  MoveL 10167 to (522.4, 527.74, 184) mm, rotated rx -180 ry 0 rz 160 deg; joints [9.235, 54.746, -7.823, -142.539, 53.417, 155.455]
  Set speed (17.9 mm/s)
  Call Extruder(893.93163)
  MoveL 10168 to (521.41, 528.51, 184) mm, rotated rx 180 ry 0 rz 160 deg; joints [9.346, 54.585, -7.526, -142.475, 53.571, 155.484]
  Set speed (17.9 mm/s)
  Call Extruder(896.88421)
  MoveL 10169 to (520.65, 529.06, 184) mm, rotated rx -180 ry 0 rz 160 deg; joints [9.426, 54.462, -7.298, -142.432, 53.688, 155.51]
  Call Extruder(901.40874)
  MoveL 10170 to (519.47, 529.87, 184) mm, rotated rx 180 ry 0 rz 160 deg; joints [9.545, 54.269, -6.939, -142.372, 53.869, 155.556]
  Call Extruder(903.78888)
  MoveL 10171 to (518.83, 530.27, 184) mm, rotated rx 180 ry 0 rz 160 deg; joints [9.606, 54.164, -6.745, -142.343, 53.965, 155.583]
  Set speed (17.9 mm/s)
  Call Extruder(906.07988)
  MoveL 10172 to (518.21, 530.65, 184) mm, rotated rx 180 ry 0 rz 160 deg; joints [9.663, 54.063, -6.556, -142.317, 54.057, 155.611]
  Call Extruder(910.83041)
  MoveL 10173 to (516.91, 531.39, 184) mm, rotated rx 180 ry 0 rz 160 deg; joints [9.779, 53.847, -6.156, -142.269, 54.25, 155.674]
  Set speed (17.8 mm/s)
  Call Extruder(914.28684)
  MoveL 10174 to (515.94, 531.89, 184) mm, rotated rx 180 ry 0 rz 160 deg; joints [9.859, 53.687, -5.859, -142.239, 54.392, 155.725]
  Call Extruder(917.59208)
  MoveL 10175 to (515, 532.34, 184) mm, rotated rx 180 ry 0 rz 160 deg; joints [9.933, 53.53, -5.568, -142.215, 54.528, 155.778]
  Set speed (17.9 mm/s)
  Call Extruder(922.23001)
  MoveL 10176 to (513.65, 532.93, 184) mm, rotated rx -180 ry 0 rz 160 deg; joints [10.032, 53.306, -5.154, -142.187, 54.719, 155.857]
  Set speed (17.9 mm/s)
  Call Extruder(926.66688)
  MoveL 10177 to (512.34, 533.45, 184) mm, rotated rx 180 ry 0 rz 160 deg; joints [10.121, 53.088, -4.749, -142.168, 54.903, 155.939]
  Set speed (17.8 mm/s)
  Call Extruder(929.18658)
  MoveL 10178 to (511.59, 533.71, 184) mm, rotated rx -180 ry 0 rz 160 deg; joints [10.169, 52.962, -4.515, -142.161, 55.008, 155.989]
  Set speed (17.8 mm/s)
  Call Extruder(932.98840)
  MoveL 10179 to (510.45, 534.08, 184) mm, rotated rx 180 ry 0 rz 160 deg; joints [10.239, 52.771, -4.161, -142.153, 55.165, 156.067]
  Set speed (17.8 mm/s)
  Call Extruder(936.81967)
  MoveL 10180 to (509.29, 534.42, 184) mm, rotated rx -180 ry 0 rz 160 deg; joints [10.305, 52.576, -3.799, -142.15, 55.323, 156.149]
  Set speed (17.8 mm/s)
  Call Extruder(940.52296)
  MoveL 10181 to (508.15, 534.7, 184) mm, rotated rx -180 ry 0 rz 160 deg; joints [10.364, 52.384, -3.444, -142.153, 55.476, 156.233]
  Set speed (17.9 mm/s)
  Call Extruder(945.30301)
  MoveL 10182 to (506.68, 535.02, 184) mm, rotated rx -180 ry 0 rz 160 deg; joints [10.436, 52.134, -2.982, -142.163, 55.673, 156.347]
  Call Extruder(949.97825)
  MoveL 10183 to (505.22, 535.27, 184) mm, rotated rx -180 ry 0 rz 160 deg; joints [10.498, 51.886, -2.524, -142.182, 55.864, 156.464]
  Set speed (17.8 mm/s)
  Call Extruder(954.40667)
  MoveL 10184 to (503.83, 535.45, 184) mm, rotated rx 180 ry 0 rz 160 deg; joints [10.552, 51.65, -2.087, -142.206, 56.044, 156.579]
  Set speed (17.9 mm/s)
  Call Extruder(959.14962)
  MoveL 10185 to (502.33, 535.57, 184) mm, rotated rx -180 ry 0 rz 160 deg; joints [10.602, 51.396, -1.616, -142.24, 56.235, 156.708]
  Set speed (17.9 mm/s)
  Call Extruder(963.82186)
  MoveL 10186 to (500.86, 535.64, 184) mm, rotated rx 180 ry 0 rz 160 deg; joints [10.644, 51.143, -1.149, -142.281, 56.421, 156.84]
  Set speed (17.9 mm/s)
  Call Extruder(968.31975)
  MoveL 10187 to (499.43, 535.65, 184) mm, rotated rx 180 ry 0 rz 160 deg; joints [10.678, 50.899, -0.698, -142.327, 56.598, 156.971]
  Set speed (10.0 mm/s)
  MoveL 10188 to (499.43, 535.65, 188) mm, rotated rx -180 ry 0 rz 160 deg; joints [10.678, 50.375, -0.656, -142.13, 56.216, 156.616]
  Set speed (120.0 mm/s)
  MoveL 10189 to (500.85, 535.22, 188) mm, rotated rx -180 ry 0 rz 160 deg; joints [10.593, 50.605, -1.079, -142.145, 56.03, 156.526]
  Set speed (18.0 mm/s)
  Call Extruder(972.66654)
  MoveL 10190 to (499.46, 535.23, 188) mm, rotated rx 180 ry 0 rz 160 deg; joints [10.625, 50.366, -0.641, -142.191, 56.201, 156.653]
  Call Extruder(977.34606)
  MoveL 10191 to (497.97, 535.17, 188) mm, rotated rx -180 ry 0 rz 160 deg; joints [10.653, 50.109, -0.168, -142.248, 56.382, 156.795]
  Set speed (18.0 mm/s)
  Call Extruder(981.88642)
  MoveL 10192 to (496.53, 535.06, 188) mm, rotated rx -180 ry 0 rz 160 deg; joints [10.673, 49.859, 0.291, -142.311, 56.555, 156.936]
  Call Extruder(986.34744)
  MoveL 10193 to (495.12, 534.89, 188) mm, rotated rx 180 ry 0 rz 160 deg; joints [10.685, 49.613, 0.741, -142.38, 56.722, 157.078]
  Set speed (18.0 mm/s)
  Call Extruder(990.84090)
  MoveL 10194 to (493.71, 534.67, 188) mm, rotated rx -180 ry 0 rz 160 deg; joints [10.69, 49.367, 1.192, -142.457, 56.886, 157.225]
  Set speed (18.0 mm/s)
  Call Extruder(995.48981)
  MoveL 10195 to (492.26, 534.37, 188) mm, rotated rx 180 ry 0 rz 160 deg; joints [10.687, 49.113, 1.658, -142.544, 57.053, 157.38]
  Set speed (18.0 mm/s)
  Call Extruder(999.88346)
  MoveL 10196 to (490.9, 534.04, 188) mm, rotated rx 180 ry 0 rz 160 deg; joints [10.678, 48.874, 2.095, -142.632, 57.207, 157.53]
  Set speed (18.0 mm/s)
  Call Extruder(1004.84592)
  MoveL 10197 to (489.39, 533.6, 188) mm, rotated rx 180 ry 0 rz 160 deg; joints [10.658, 48.607, 2.585, -142.74, 57.376, 157.702]
  Set speed (18.0 mm/s)
  Call Extruder(1008.82941)
  MoveL 10198 to (488.18, 533.19, 188) mm, rotated rx 180 ry 0 rz 160 deg; joints [10.635, 48.394, 2.974, -142.833, 57.509, 157.842]
  Set speed (18.0 mm/s)
  Call Extruder(1013.42678)
  MoveL 10199 to (486.82, 532.67, 188) mm, rotated rx 180 ry 0 rz 160 deg; joints [10.602, 48.151, 3.419, -142.947, 57.657, 158.005]
  Set speed (18.0 mm/s)
  Call Extruder(1017.94180)
  MoveL 10200 to (485.49, 532.11, 188) mm, rotated rx -180 ry 0 rz 160 deg; joints [10.562, 47.915, 3.851, -143.066, 57.798, 158.168]
  Set speed (17.9 mm/s)
  Call Extruder(1021.37830)
  MoveL 10201 to (484.5, 531.64, 188) mm, rotated rx -180 ry 0 rz 160 deg; joints [10.526, 47.738, 4.174, -143.16, 57.902, 158.293]
  Set speed (18.0 mm/s)
  Call Extruder(1024.92138)
  MoveL 10202 to (483.5, 531.14, 188) mm, rotated rx 180 ry 0 rz 160 deg; joints [10.485, 47.557, 4.505, -143.261, 58.007, 158.423]
  Set speed (18.0 mm/s)
  Call Extruder(1029.79745)
  MoveL 10203 to (482.14, 530.37, 188) mm, rotated rx 180 ry 0 rz 160 deg; joints [10.419, 47.313, 4.952, -143.408, 58.145, 158.603]
  Set speed (18.0 mm/s)
  Call Extruder(1034.30455)
  MoveL 10204 to (480.92, 529.62, 188) mm, rotated rx 180 ry 0 rz 160 deg; joints [10.351, 47.091, 5.356, -143.551, 58.267, 158.771]
  Call Extruder(1038.31068)
  MoveL 10205 to (479.86, 528.91, 188) mm, rotated rx -180 ry 0 rz 160 deg; joints [10.284, 46.898, 5.709, -143.682, 58.371, 158.92]
  Set speed (18.0 mm/s)
  Call Extruder(1040.61575)
  MoveL 10206 to (479.26, 528.48, 188) mm, rotated rx 180 ry 0 rz 160 deg; joints [10.243, 46.788, 5.909, -143.76, 58.43, 159.006]
  Set speed (18.0 mm/s)
  Call Extruder(1042.87029)
  MoveL 10207 to (478.69, 528.06, 188) mm, rotated rx 180 ry 0 rz 160 deg; joints [10.201, 46.682, 6.102, -143.838, 58.485, 159.091]
  Call Extruder(1045.13772)
  MoveL 10208 to (478.12, 527.61, 188) mm, rotated rx -180 ry 0 rz 160 deg; joints [10.157, 46.577, 6.294, -143.918, 58.539, 159.176]
  Set speed (18.0 mm/s)
  Call Extruder(1047.91484)
  MoveL 10209 to (477.43, 527.06, 188) mm, rotated rx 180 ry 0 rz 160 deg; joints [10.1, 46.45, 6.525, -144.017, 58.604, 159.281]
  Set speed (18.0 mm/s)
  Call Extruder(1050.88641)
  MoveL 10210 to (476.71, 526.44, 188) mm, rotated rx -180 ry 0 rz 160 deg; joints [10.037, 46.317, 6.768, -144.126, 58.67, 159.392]
  Set speed (18.0 mm/s)
  Call Extruder(1054.07637)
  MoveL 10211 to (475.96, 525.76, 188) mm, rotated rx 180 ry 0 rz 160 deg; joints [9.965, 46.177, 7.023, -144.246, 58.738, 159.512]
  Set speed (18.0 mm/s)
  Call Extruder(1056.93409)
  MoveL 10212 to (475.31, 525.13, 188) mm, rotated rx -180 ry 0 rz 160 deg; joints [9.898, 46.054, 7.247, -144.355, 58.797, 159.619]
  Set speed (18.0 mm/s)
  Call Extruder(1060.97638)
  MoveL 10213 to (474.4, 524.21, 188) mm, rotated rx -180 ry 0 rz 160 deg; joints [9.798, 45.884, 7.557, -144.514, 58.876, 159.771]
  Set speed (18.0 mm/s)
  Call Extruder(1063.75696)
  MoveL 10214 to (473.8, 523.56, 188) mm, rotated rx 180 ry 0 rz 160 deg; joints [9.726, 45.77, 7.764, -144.626, 58.927, 159.875]
  Set speed (18.0 mm/s)
  Call Extruder(1066.38918)
  MoveL 10215 to (473.25, 522.93, 188) mm, rotated rx -180 ry 0 rz 160 deg; joints [9.655, 45.664, 7.957, -144.733, 58.974, 159.973]
  Call Extruder(1070.04487)
  MoveL 10216 to (472.51, 522.03, 188) mm, rotated rx 180 ry 0 rz 160 deg; joints [9.554, 45.522, 8.216, -144.885, 59.034, 160.109]
  Set speed (18.0 mm/s)
  Call Extruder(1074.65991)
  MoveL 10217 to (471.61, 520.87, 188) mm, rotated rx 180 ry 0 rz 160 deg; joints [9.419, 45.348, 8.532, -145.081, 59.105, 160.28]
  Set speed (18.0 mm/s)
  Call Extruder(1076.75495)
  MoveL 10218 to (471.22, 520.33, 188) mm, rotated rx -180 ry 0 rz 160 deg; joints [9.356, 45.272, 8.67, -145.172, 59.135, 160.357]
  Set speed (18.0 mm/s)
  Call Extruder(1079.16479)
  MoveL 10219 to (470.78, 519.69, 188) mm, rotated rx 180 ry 0 rz 160 deg; joints [9.282, 45.187, 8.826, -145.277, 59.168, 160.445]
  Set speed (18.0 mm/s)
  Call Extruder(1081.78892)
  MoveL 10220 to (470.33, 519, 188) mm, rotated rx 180 ry 0 rz 160 deg; joints [9.199, 45.096, 8.991, -145.393, 59.201, 160.541]
  Set speed (18.0 mm/s)
  Call Extruder(1083.58163)
  MoveL 10221 to (470.02, 518.51, 188) mm, rotated rx -180 ry 0 rz 160 deg; joints [9.141, 45.036, 9.1, -145.474, 59.222, 160.606]
  Set speed (18.0 mm/s)
  Call Extruder(1086.37228)
  MoveL 10222 to (469.57, 517.75, 188) mm, rotated rx 180 ry 0 rz 160 deg; joints [9.049, 44.944, 9.267, -145.6, 59.254, 160.707]
  Set speed (18.0 mm/s)
  Call Extruder(1090.55089)
  MoveL 10223 to (468.91, 516.59, 188) mm, rotated rx -180 ry 0 rz 160 deg; joints [8.908, 44.812, 9.506, -145.791, 59.296, 160.857]
  Call Extruder(1092.71321)
  MoveL 10224 to (468.6, 515.98, 188) mm, rotated rx 180 ry 0 rz 160 deg; joints [8.833, 44.747, 9.625, -145.891, 59.315, 160.934]
  Set speed (18.0 mm/s)
  Call Extruder(1094.90666)
  MoveL 10225 to (468.29, 515.35, 188) mm, rotated rx -180 ry 0 rz 160 deg; joints [8.755, 44.683, 9.741, -145.994, 59.334, 161.011]
  Call Extruder(1099.61642)
  MoveL 10226 to (467.66, 513.99, 188) mm, rotated rx 180 ry 0 rz 160 deg; joints [8.585, 44.552, 9.979, -146.216, 59.367, 161.176]
  Call Extruder(1103.98776)
  MoveL 10227 to (467.14, 512.7, 188) mm, rotated rx 180 ry 0 rz 160 deg; joints [8.423, 44.439, 10.185, -146.425, 59.392, 161.327]
  Set speed (18.0 mm/s)
  Call Extruder(1108.45870)
  MoveL 10228 to (466.65, 511.36, 188) mm, rotated rx -180 ry 0 rz 160 deg; joints [8.252, 44.332, 10.379, -146.642, 59.41, 161.478]
  Set speed (18.0 mm/s)
  Call Extruder(1110.08883)
  MoveL 10229 to (466.49, 510.87, 188) mm, rotated rx 180 ry 0 rz 160 deg; joints [8.189, 44.295, 10.446, -146.721, 59.415, 161.533]
  Set speed (17.9 mm/s)
  Call Extruder(1113.55157)
  MoveL 10230 to (466.16, 509.82, 188) mm, rotated rx 180 ry 0 rz 160 deg; joints [8.053, 44.22, 10.581, -146.891, 59.423, 161.648]
  Set speed (18.0 mm/s)
  Call Extruder(1117.54079)
  MoveL 10231 to (465.83, 508.59, 188) mm, rotated rx -180 ry 0 rz 160 deg; joints [7.893, 44.141, 10.724, -147.087, 59.427, 161.778]
  Set speed (18.0 mm/s)
  Call Extruder(1122.08861)
  MoveL 10232 to (465.51, 507.18, 188) mm, rotated rx 180 ry 0 rz 160 deg; joints [7.708, 44.06, 10.871, -147.313, 59.425, 161.923]
  Set speed (18.0 mm/s)
  Call Extruder(1126.74925)
  MoveL 10233 to (465.23, 505.72, 188) mm, rotated rx -180 ry 0 rz 160 deg; joints [7.515, 43.987, 11.004, -147.545, 59.415, 162.069]
  Set speed (18.0 mm/s)
  Call Extruder(1131.27133)
  MoveL 10234 to (465.03, 504.3, 188) mm, rotated rx 180 ry 0 rz 160 deg; joints [7.325, 43.926, 11.115, -147.771, 59.399, 162.207]
  Call Extruder(1135.79933)
  MoveL 10235 to (464.88, 502.87, 188) mm, rotated rx 180 ry 0 rz 160 deg; joints [7.132, 43.875, 11.208, -147.997, 59.375, 162.341]
  Call Extruder(1140.43813)
  MoveL 10236 to (464.8, 501.39, 188) mm, rotated rx -180 ry 0 rz 160 deg; joints [6.933, 43.832, 11.284, -148.229, 59.344, 162.475]
  Set speed (17.9 mm/s)
  Call Extruder(1144.77516)
  MoveL 10237 to (464.77, 500.01, 188) mm, rotated rx -180 ry 0 rz 160 deg; joints [6.745, 43.802, 11.339, -148.445, 59.309, 162.596]
  Set speed (17.9 mm/s)
  Call Extruder(1148.91787)
  MoveL 10238 to (464.79, 498.69, 188) mm, rotated rx 180 ry 0 rz 160 deg; joints [6.565, 43.782, 11.376, -148.65, 59.269, 162.708]
  Set speed (18.0 mm/s)
  Call Extruder(1152.91329)
  MoveL 10239 to (464.86, 497.43, 188) mm, rotated rx 180 ry 0 rz 160 deg; joints [6.39, 43.77, 11.397, -148.847, 59.226, 162.813]
  Set speed (18.0 mm/s)
  Call Extruder(1156.99605)
  MoveL 10240 to (464.98, 496.13, 188) mm, rotated rx 180 ry 0 rz 160 deg; joints [6.211, 43.766, 11.404, -149.047, 59.176, 162.917]
  Set speed (18.0 mm/s)
  Call Extruder(1161.07084)
  MoveL 10241 to (465.15, 494.84, 188) mm, rotated rx 180 ry 0 rz 160 deg; joints [6.033, 43.771, 11.396, -149.244, 59.12, 163.017]
  Call Extruder(1164.98026)
  MoveL 10242 to (465.35, 493.61, 188) mm, rotated rx -180 ry 0 rz 160 deg; joints [5.862, 43.783, 11.374, -149.432, 59.062, 163.109]
  Set speed (18.0 mm/s)
  Call Extruder(1169.18292)
  MoveL 10243 to (465.62, 492.3, 188) mm, rotated rx 180 ry 0 rz 160 deg; joints [5.679, 43.804, 11.336, -149.631, 58.994, 163.204]
  Set speed (18.0 mm/s)
  Call Extruder(1173.28818)
  MoveL 10244 to (465.93, 491.03, 188) mm, rotated rx -180 ry 0 rz 160 deg; joints [5.502, 43.833, 11.284, -149.822, 58.923, 163.292]
  Set speed (18.0 mm/s)
  Call Extruder(1177.30378)
  MoveL 10245 to (466.27, 489.8, 188) mm, rotated rx 180 ry 0 rz 160 deg; joints [5.329, 43.869, 11.218, -150.007, 58.848, 163.375]
  Set speed (18.0 mm/s)
  Call Extruder(1181.38217)
  MoveL 10246 to (466.67, 488.57, 188) mm, rotated rx 180 ry 0 rz 160 deg; joints [5.155, 43.914, 11.137, -150.19, 58.767, 163.454]
  Call Extruder(1185.55335)
  MoveL 10247 to (467.13, 487.32, 188) mm, rotated rx -180 ry 0 rz 160 deg; joints [4.979, 43.968, 11.038, -150.375, 58.678, 163.531]
  Set speed (18.0 mm/s)
  Call Extruder(1189.67180)
  MoveL 10248 to (467.62, 486.11, 188) mm, rotated rx -180 ry 0 rz 160 deg; joints [4.807, 44.03, 10.927, -150.552, 58.586, 163.603]
  Set speed (18.0 mm/s)
  Call Extruder(1193.68830)
  MoveL 10249 to (468.15, 484.94, 188) mm, rotated rx 180 ry 0 rz 160 deg; joints [4.642, 44.097, 10.805, -150.721, 58.492, 163.668]
  Set speed (18.0 mm/s)
  Call Extruder(1197.78489)
  MoveL 10250 to (468.73, 483.77, 188) mm, rotated rx 180 ry 0 rz 160 deg; joints [4.477, 44.174, 10.665, -150.889, 58.391, 163.73]
  Set speed (18.0 mm/s)
  Call Extruder(1201.93796)
  MoveL 10251 to (469.36, 482.61, 188) mm, rotated rx 180 ry 0 rz 160 deg; joints [4.312, 44.259, 10.51, -151.054, 58.284, 163.788]
  Set speed (17.9 mm/s)
  Call Extruder(1206.52795)
  MoveL 10252 to (470.1, 481.36, 188) mm, rotated rx 180 ry 0 rz 160 deg; joints [4.134, 44.363, 10.323, -151.23, 58.161, 163.846]
  Set speed (18.0 mm/s)
  Call Extruder(1209.83621)
  MoveL 10253 to (470.68, 480.47, 188) mm, rotated rx -180 ry 0 rz 160 deg; joints [4.008, 44.443, 10.176, -151.353, 58.068, 163.884]
  Set speed (18.0 mm/s)
  Call Extruder(1214.03556)
  MoveL 10254 to (471.44, 479.37, 188) mm, rotated rx -180 ry 0 rz 160 deg; joints [3.852, 44.552, 9.978, -151.503, 57.947, 163.928]
  Set speed (18.0 mm/s)
  Call Extruder(1218.05006)
  MoveL 10255 to (472.21, 478.35, 188) mm, rotated rx -180 ry 0 rz 160 deg; joints [3.707, 44.664, 9.776, -151.641, 57.827, 163.964]
  Call Extruder(1222.27088)
  MoveL 10256 to (473.05, 477.31, 188) mm, rotated rx 180 ry 0 rz 160 deg; joints [3.558, 44.788, 9.551, -151.779, 57.696, 163.997]
  Set speed (18.0 mm/s)
  Call Extruder(1226.25255)
  MoveL 10257 to (473.88, 476.35, 188) mm, rotated rx 180 ry 0 rz 160 deg; joints [3.423, 44.911, 9.326, -151.904, 57.57, 164.024]
  Call Extruder(1230.41361)
  MoveL 10258 to (474.79, 475.39, 188) mm, rotated rx -180 ry 0 rz 160 deg; joints [3.285, 45.047, 9.079, -152.027, 57.434, 164.046]
  Set speed (18.0 mm/s)
  Call Extruder(1234.40312)
  MoveL 10259 to (475.7, 474.49, 188) mm, rotated rx 180 ry 0 rz 160 deg; joints [3.158, 45.184, 8.83, -152.138, 57.3, 164.062]
  Set speed (18.0 mm/s)
  Call Extruder(1238.47932)
  MoveL 10260 to (476.65, 473.62, 188) mm, rotated rx 180 ry 0 rz 160 deg; joints [3.034, 45.33, 8.565, -152.245, 57.16, 164.073]
  Set speed (18.0 mm/s)
  Call Extruder(1242.64814)
  MoveL 10261 to (477.66, 472.75, 188) mm, rotated rx -180 ry 0 rz 160 deg; joints [2.911, 45.485, 8.282, -152.347, 57.014, 164.078]
  Set speed (18.0 mm/s)
  Call Extruder(1247.06946)
  MoveL 10262 to (478.77, 471.88, 188) mm, rotated rx -180 ry 0 rz 160 deg; joints [2.788, 45.657, 7.97, -152.446, 56.856, 164.078]
  Call Extruder(1250.74658)
  MoveL 10263 to (479.71, 471.2, 188) mm, rotated rx 180 ry 0 rz 160 deg; joints [2.69, 45.805, 7.701, -152.522, 56.721, 164.073]
  Set speed (18.0 mm/s)
  Call Extruder(1254.67182)
  MoveL 10264 to (480.75, 470.49, 188) mm, rotated rx -180 ry 0 rz 160 deg; joints [2.59, 45.967, 7.405, -152.597, 56.576, 164.062]
  Call Extruder(1258.92817)
  MoveL 10265 to (481.9, 469.78, 188) mm, rotated rx 180 ry 0 rz 160 deg; joints [2.488, 46.149, 7.074, -152.669, 56.415, 164.045]
  Call Extruder(1263.01389)
  MoveL 10266 to (483.02, 469.13, 188) mm, rotated rx 180 ry 0 rz 160 deg; joints [2.396, 46.329, 6.747, -152.73, 56.258, 164.023]
  Set speed (18.0 mm/s)
  Call Extruder(1266.90627)
  MoveL 10267 to (484.12, 468.55, 188) mm, rotated rx 180 ry 0 rz 160 deg; joints [2.313, 46.504, 6.427, -152.781, 56.107, 163.996]
  Set speed (18.0 mm/s)
  Call Extruder(1271.14857)
  MoveL 10268 to (485.34, 467.96, 188) mm, rotated rx 180 ry 0 rz 160 deg; joints [2.23, 46.7, 6.07, -152.828, 55.941, 163.961]
  Set speed (18.0 mm/s)
  Call Extruder(1275.23430)
  MoveL 10269 to (486.53, 467.45, 188) mm, rotated rx 180 ry 0 rz 160 deg; joints [2.155, 46.893, 5.718, -152.866, 55.779, 163.922]
  Set speed (18.0 mm/s)
  Call Extruder(1279.11549)
  MoveL 10270 to (487.68, 466.99, 188) mm, rotated rx 180 ry 0 rz 160 deg; joints [2.09, 47.08, 5.376, -152.893, 55.623, 163.88]
  Set speed (18.0 mm/s)
  Call Extruder(1283.35551)
  MoveL 10271 to (488.95, 466.54, 188) mm, rotated rx -180 ry 0 rz 160 deg; joints [2.026, 47.288, 4.996, -152.914, 55.452, 163.827]
  Call Extruder(1287.41205)
  MoveL 10272 to (490.19, 466.16, 188) mm, rotated rx 180 ry 0 rz 160 deg; joints [1.971, 47.491, 4.626, -152.926, 55.288, 163.771]
  Set speed (18.0 mm/s)
  Call Extruder(1291.52994)
  MoveL 10273 to (491.45, 465.82, 188) mm, rotated rx 180 ry 0 rz 160 deg; joints [1.921, 47.7, 4.244, -152.93, 55.12, 163.708]
  Call Extruder(1295.44431)
  MoveL 10274 to (492.67, 465.54, 188) mm, rotated rx -180 ry 0 rz 160 deg; joints [1.879, 47.902, 3.875, -152.926, 54.959, 163.644]
  Call Extruder(1299.59154)
  MoveL 10275 to (493.96, 465.29, 188) mm, rotated rx 180 ry 0 rz 160 deg; joints [1.841, 48.118, 3.48, -152.913, 54.789, 163.57]
  Set speed (18.0 mm/s)
  Call Extruder(1303.53526)
  MoveL 10276 to (495.2, 465.09, 188) mm, rotated rx 180 ry 0 rz 160 deg; joints [1.811, 48.326, 3.099, -152.893, 54.627, 163.494]
  Set speed (18.0 mm/s)
  Call Extruder(1307.77538)
  MoveL 10277 to (496.55, 464.94, 188) mm, rotated rx 180 ry 0 rz 160 deg; joints [1.785, 48.552, 2.686, -152.862, 54.452, 163.406]
  Call Extruder(1311.80226)
  MoveL 10278 to (497.82, 464.84, 188) mm, rotated rx 180 ry 0 rz 160 deg; joints [1.767, 48.768, 2.289, -152.825, 54.287, 163.318]
  Set speed (18.0 mm/s)
  Call Extruder(1315.97904)
  MoveL 10279 to (499.15, 464.78, 188) mm, rotated rx 180 ry 0 rz 160 deg; joints [1.755, 48.995, 1.875, -152.777, 54.116, 163.22]
  Set speed (18.0 mm/s)
  Call Extruder(1319.97418)
  MoveL 10280 to (500.42, 464.77, 188) mm, rotated rx -180 ry 0 rz 160 deg; joints [1.748, 49.212, 1.476, -152.724, 53.953, 163.122]
  Call Extruder(1324.11243)
  MoveL 10281 to (501.74, 464.81, 188) mm, rotated rx 180 ry 0 rz 160 deg; joints [1.748, 49.439, 1.061, -152.661, 53.786, 163.015]
  Set speed (18.0 mm/s)
  Call Extruder(1328.11577)
  MoveL 10282 to (503.01, 464.9, 188) mm, rotated rx -180 ry 0 rz 160 deg; joints [1.754, 49.658, 0.658, -152.592, 53.625, 162.906]
  Set speed (18.0 mm/s)
  Call Extruder(1332.26885)
  MoveL 10283 to (504.33, 465.04, 188) mm, rotated rx -180 ry 0 rz 160 deg; joints [1.767, 49.887, 0.239, -152.512, 53.459, 162.788]
  Set speed (18.0 mm/s)
  Call Extruder(1336.19152)
  MoveL 10284 to (505.56, 465.21, 188) mm, rotated rx 180 ry 0 rz 160 deg; joints [1.784, 50.103, -0.157, -152.43, 53.305, 162.672]
  Set speed (18.0 mm/s)
  Call Extruder(1340.36875)
  MoveL 10285 to (506.87, 465.44, 188) mm, rotated rx 180 ry 0 rz 160 deg; joints [1.808, 50.333, -0.579, -152.334, 53.142, 162.544]
  Set speed (18.0 mm/s)
  Call Extruder(1344.45433)
  MoveL 10286 to (508.14, 465.72, 188) mm, rotated rx 180 ry 0 rz 160 deg; joints [1.838, 50.557, -0.991, -152.233, 52.984, 162.413]
  Call Extruder(1348.38804)
  MoveL 10287 to (509.36, 466.03, 188) mm, rotated rx 180 ry 0 rz 160 deg; joints [1.872, 50.772, -1.387, -152.129, 52.835, 162.283]
  Set speed (18.0 mm/s)
  Call Extruder(1352.55747)
  MoveL 10288 to (510.63, 466.41, 188) mm, rotated rx 180 ry 0 rz 160 deg; joints [1.914, 51, -1.805, -152.011, 52.679, 162.141]
  Call Extruder(1356.69366)
  MoveL 10289 to (511.88, 466.83, 188) mm, rotated rx -180 ry 0 rz 160 deg; joints [1.961, 51.224, -2.217, -151.887, 52.528, 161.995]
  Set speed (18.0 mm/s)
  Call Extruder(1360.78521)
  MoveL 10290 to (513.1, 467.29, 188) mm, rotated rx 180 ry 0 rz 160 deg; joints [2.013, 51.444, -2.622, -151.758, 52.381, 161.847]
  Set speed (18.0 mm/s)
  Call Extruder(1364.85814)
  MoveL 10291 to (514.29, 467.8, 188) mm, rotated rx -180 ry 0 rz 160 deg; joints [2.07, 51.661, -3.022, -151.623, 52.239, 161.696]
  Set speed (18.0 mm/s)
  Call Extruder(1368.90731)
  MoveL 10292 to (515.46, 468.34, 188) mm, rotated rx -180 ry 0 rz 160 deg; joints [2.132, 51.875, -3.415, -151.482, 52.1, 161.542]
  Set speed (18.0 mm/s)
  Call Extruder(1373.11651)
  MoveL 10293 to (516.65, 468.95, 188) mm, rotated rx -180 ry 0 rz 160 deg; joints [2.201, 52.095, -3.819, -151.329, 51.96, 161.379]
  Set speed (18.0 mm/s)
  Call Extruder(1376.93125)
  MoveL 10294 to (517.71, 469.55, 188) mm, rotated rx -180 ry 0 rz 160 deg; joints [2.269, 52.291, -4.181, -151.186, 51.837, 161.227]
  Set speed (18.0 mm/s)
  Call Extruder(1380.94465)
  MoveL 10295 to (518.81, 470.21, 188) mm, rotated rx -180 ry 0 rz 160 deg; joints [2.345, 52.495, -4.556, -151.029, 51.711, 161.065]
  Set speed (18.0 mm/s)
  Call Extruder(1385.22698)
  MoveL 10296 to (519.95, 470.96, 188) mm, rotated rx 180 ry 0 rz 160 deg; joints [2.43, 52.709, -4.951, -150.856, 51.582, 160.889]
  Set speed (18.0 mm/s)
  Call Extruder(1389.19566)
  MoveL 10297 to (520.97, 471.69, 188) mm, rotated rx 180 ry 0 rz 160 deg; joints [2.514, 52.904, -5.31, -150.692, 51.466, 160.724]
  Set speed (18.0 mm/s)
  Call Extruder(1393.20228)
  MoveL 10298 to (521.98, 472.47, 188) mm, rotated rx 180 ry 0 rz 160 deg; joints [2.604, 53.096, -5.665, -150.52, 51.354, 160.555]
  Set speed (18.0 mm/s)
  Call Extruder(1397.53386)
  MoveL 10299 to (523.05, 473.35, 188) mm, rotated rx -180 ry 0 rz 160 deg; joints [2.704, 53.301, -6.042, -150.33, 51.237, 160.37]
  Call Extruder(1401.51926)
  MoveL 10300 to (523.99, 474.2, 188) mm, rotated rx -180 ry 0 rz 160 deg; joints [2.801, 53.484, -6.38, -150.151, 51.136, 160.198]
  Set speed (18.0 mm/s)
  Call Extruder(1405.45304)
  MoveL 10301 to (524.89, 475.07, 188) mm, rotated rx 180 ry 0 rz 160 deg; joints [2.901, 53.66, -6.705, -149.971, 51.041, 160.027]
  Call Extruder(1408.20491)
  MoveL 10302 to (525.5, 475.7, 188) mm, rotated rx 180 ry 0 rz 160 deg; joints [2.973, 53.781, -6.927, -149.843, 50.977, 159.906]
  Call Extruder(1412.73519)
  MoveL 10303 to (526.48, 476.76, 188) mm, rotated rx 180 ry 0 rz 160 deg; joints [3.094, 53.974, -7.285, -149.629, 50.878, 159.707]
  Call Extruder(1414.45387)
  MoveL 10304 to (526.84, 477.17, 188) mm, rotated rx 180 ry 0 rz 160 deg; joints [3.141, 54.046, -7.417, -149.547, 50.842, 159.632]
  Set speed (18.0 mm/s)
  Call Extruder(1417.26422)
  MoveL 10305 to (527.41, 477.86, 188) mm, rotated rx 180 ry 0 rz 160 deg; joints [3.22, 54.161, -7.629, -149.411, 50.785, 159.508]
  Set speed (18.0 mm/s)
  Call Extruder(1419.02542)
  MoveL 10306 to (527.76, 478.3, 188) mm, rotated rx -180 ry 0 rz 160 deg; joints [3.271, 54.231, -7.759, -149.326, 50.752, 159.43]
  Set speed (18.0 mm/s)
  Call Extruder(1422.62788)
  MoveL 10307 to (528.45, 479.22, 188) mm, rotated rx -180 ry 0 rz 160 deg; joints [3.375, 54.373, -8.021, -149.149, 50.685, 159.271]
  Call Extruder(1425.90342)
  MoveL 10308 to (529.05, 480.07, 188) mm, rotated rx -180 ry 0 rz 160 deg; joints [3.473, 54.497, -8.249, -148.987, 50.63, 159.126]
  Set speed (18.0 mm/s)
  Call Extruder(1430.31031)
  MoveL 10309 to (529.82, 481.24, 188) mm, rotated rx -180 ry 0 rz 160 deg; joints [3.607, 54.657, -8.546, -148.767, 50.562, 158.932]
  Call Extruder(1432.57231)
  MoveL 10310 to (530.2, 481.86, 188) mm, rotated rx -180 ry 0 rz 160 deg; joints [3.677, 54.737, -8.693, -148.653, 50.529, 158.833]
  Set speed (18.0 mm/s)
  Call Extruder(1434.85297)
  MoveL 10311 to (530.57, 482.48, 188) mm, rotated rx 180 ry 0 rz 160 deg; joints [3.749, 54.815, -8.838, -148.538, 50.499, 158.733]
  Set speed (18.0 mm/s)
  Call Extruder(1437.54318)
  MoveL 10312 to (530.98, 483.23, 188) mm, rotated rx 180 ry 0 rz 160 deg; joints [3.834, 54.905, -9.003, -148.402, 50.465, 158.616]
  Set speed (18.0 mm/s)
  Call Extruder(1440.05996)
  MoveL 10313 to (531.36, 483.94, 188) mm, rotated rx -180 ry 0 rz 160 deg; joints [3.916, 54.985, -9.152, -148.274, 50.437, 158.507]
  Set speed (18.0 mm/s)
  Call Extruder(1443.80508)
  MoveL 10314 to (531.88, 485.01, 188) mm, rotated rx 180 ry 0 rz 160 deg; joints [4.038, 55.101, -9.367, -148.084, 50.398, 158.345]
  Set speed (18.0 mm/s)
  Call Extruder(1446.17698)
  MoveL 10315 to (532.2, 485.7, 188) mm, rotated rx 180 ry 0 rz 160 deg; joints [4.117, 55.171, -9.496, -147.963, 50.377, 158.244]
  Set speed (18.0 mm/s)
  Call Extruder(1450.65174)
  MoveL 10316 to (532.75, 487.01, 188) mm, rotated rx 180 ry 0 rz 160 deg; joints [4.268, 55.296, -9.727, -147.734, 50.343, 158.055]
  Set speed (18.0 mm/s)
  Call Extruder(1455.23639)
  MoveL 10317 to (533.26, 488.38, 188) mm, rotated rx 180 ry 0 rz 160 deg; joints [4.424, 55.416, -9.948, -147.5, 50.316, 157.864]
  Set speed (18.0 mm/s)
  Call Extruder(1459.76952)
  MoveL 10318 to (533.71, 489.75, 188) mm, rotated rx 180 ry 0 rz 160 deg; joints [4.582, 55.523, -10.147, -147.27, 50.299, 157.678]
  Set speed (18.0 mm/s)
  Call Extruder(1464.25238)
  MoveL 10319 to (534.1, 491.13, 188) mm, rotated rx -180 ry 0 rz 160 deg; joints [4.74, 55.621, -10.327, -147.042, 50.29, 157.499]
  Set speed (18.0 mm/s)
  Call Extruder(1468.82912)
  MoveL 10320 to (534.44, 492.54, 188) mm, rotated rx 180 ry 0 rz 160 deg; joints [4.904, 55.71, -10.493, -146.812, 50.289, 157.319]
  Set speed (18.0 mm/s)
  Call Extruder(1473.37678)
  MoveL 10321 to (534.71, 493.96, 188) mm, rotated rx 180 ry 0 rz 160 deg; joints [5.068, 55.788, -10.638, -146.585, 50.297, 157.146]
  Set speed (18.0 mm/s)
  Call Extruder(1477.89060)
  MoveL 10322 to (534.93, 495.39, 188) mm, rotated rx 180 ry 0 rz 160 deg; joints [5.232, 55.856, -10.763, -146.361, 50.313, 156.979]
  Call Extruder(1482.51856)
  MoveL 10323 to (535.09, 496.85, 188) mm, rotated rx 180 ry 0 rz 160 deg; joints [5.402, 55.914, -10.87, -146.135, 50.338, 156.814]
  Set speed (18.0 mm/s)
  Call Extruder(1486.96125)
  MoveL 10324 to (535.19, 498.26, 188) mm, rotated rx -180 ry 0 rz 160 deg; joints [5.567, 55.96, -10.956, -145.921, 50.371, 156.66]
  Set speed (18.0 mm/s)
  Call Extruder(1491.46924)
  MoveL 10325 to (535.23, 499.7, 188) mm, rotated rx -180 ry 0 rz 160 deg; joints [5.734, 55.997, -11.023, -145.707, 50.412, 156.511]
  Set speed (18.0 mm/s)
  Call Extruder(1496.08278)
  MoveL 10326 to (535.21, 501.17, 188) mm, rotated rx -180 ry 0 rz 160 deg; joints [5.906, 56.022, -11.071, -145.492, 50.463, 156.364]
  Set speed (18.0 mm/s)
  Call Extruder(1500.51812)
  MoveL 10327 to (535.14, 502.58, 188) mm, rotated rx -180 ry 0 rz 160 deg; joints [6.072, 56.037, -11.097, -145.29, 50.519, 156.23]
  Set speed (18.0 mm/s)
  Call Extruder(1505.03782)
  MoveL 10328 to (535, 504.01, 188) mm, rotated rx -180 ry 0 rz 160 deg; joints [6.242, 56.04, -11.104, -145.088, 50.585, 156.1]
  Call Extruder(1509.65812)
  MoveL 10329 to (534.8, 505.47, 188) mm, rotated rx 180 ry 0 rz 160 deg; joints [6.415, 56.033, -11.091, -144.886, 50.66, 155.975]
  Set speed (18.0 mm/s)
  Call Extruder(1514.02191)
  MoveL 10330 to (534.56, 506.84, 188) mm, rotated rx 180 ry 0 rz 160 deg; joints [6.578, 56.016, -11.059, -144.7, 50.739, 155.864]
  Set speed (18.0 mm/s)
  Call Extruder(1518.75011)
  MoveL 10331 to (534.24, 508.31, 188) mm, rotated rx -180 ry 0 rz 160 deg; joints [6.754, 55.987, -11.004, -144.505, 50.832, 155.751]
  Set speed (18.0 mm/s)
  Call Extruder(1523.16134)
  MoveL 10332 to (533.88, 509.67, 188) mm, rotated rx 180 ry 0 rz 160 deg; joints [6.918, 55.948, -10.934, -144.328, 50.925, 155.654]
  Set speed (18.0 mm/s)
  Call Extruder(1527.51477)
  MoveL 10333 to (533.47, 510.99, 188) mm, rotated rx 180 ry 0 rz 160 deg; joints [7.079, 55.9, -10.845, -144.158, 51.025, 155.566]
  Set speed (18.0 mm/s)
  Call Extruder(1532.12317)
  MoveL 10334 to (532.98, 512.38, 188) mm, rotated rx -180 ry 0 rz 160 deg; joints [7.248, 55.839, -10.731, -143.986, 51.137, 155.482]
  Set speed (18.0 mm/s)
  Call Extruder(1534.50980)
  MoveL 10335 to (532.71, 513.08, 188) mm, rotated rx 180 ry 0 rz 160 deg; joints [7.335, 55.803, -10.665, -143.898, 51.198, 155.441]
  Set speed (18.0 mm/s)
  Call Extruder(1536.63986)
  MoveL 10336 to (532.46, 513.71, 188) mm, rotated rx -180 ry 0 rz 160 deg; joints [7.412, 55.769, -10.602, -143.822, 51.253, 155.406]
  Set speed (18.0 mm/s)
  Call Extruder(1541.36975)
  MoveL 10337 to (531.84, 515.09, 188) mm, rotated rx 180 ry 0 rz 160 deg; joints [7.582, 55.685, -10.446, -143.657, 51.382, 155.336]
  Call Extruder(1545.64749)
  MoveL 10338 to (531.23, 516.31, 188) mm, rotated rx -180 ry 0 rz 160 deg; joints [7.735, 55.599, -10.286, -143.515, 51.505, 155.282]
  Set speed (18.0 mm/s)
  Call Extruder(1547.98981)
  MoveL 10339 to (530.88, 516.97, 188) mm, rotated rx -180 ry 0 rz 160 deg; joints [7.817, 55.548, -10.192, -143.44, 51.574, 155.255]
  Call Extruder(1552.40635)
  MoveL 10340 to (530.18, 518.19, 188) mm, rotated rx 180 ry 0 rz 160 deg; joints [7.972, 55.445, -10.003, -143.302, 51.709, 155.21]
  Set speed (18.0 mm/s)
  Call Extruder(1554.78510)
  MoveL 10341 to (529.78, 518.83, 188) mm, rotated rx -180 ry 0 rz 160 deg; joints [8.054, 55.386, -9.893, -143.231, 51.783, 155.19]
  Set speed (18.0 mm/s)
  Call Extruder(1557.02351)
  MoveL 10342 to (529.39, 519.43, 188) mm, rotated rx 180 ry 0 rz 160 deg; joints [8.13, 55.328, -9.786, -143.166, 51.855, 155.173]
  Call Extruder(1559.76172)
  MoveL 10343 to (528.9, 520.15, 188) mm, rotated rx -180 ry 0 rz 160 deg; joints [8.223, 55.254, -9.649, -143.088, 51.944, 155.155]
  Set speed (18.0 mm/s)
  Call Extruder(1561.55876)
  MoveL 10344 to (528.57, 520.62, 188) mm, rotated rx 180 ry 0 rz 160 deg; joints [8.284, 55.203, -9.555, -143.039, 52.004, 155.145]
  Call Extruder(1566.35721)
  MoveL 10345 to (527.65, 521.84, 188) mm, rotated rx 180 ry 0 rz 160 deg; joints [8.443, 55.061, -9.293, -142.912, 52.167, 155.124]
  Call Extruder(1570.72889)
  MoveL 10346 to (526.77, 522.91, 188) mm, rotated rx 180 ry 0 rz 160 deg; joints [8.585, 54.924, -9.038, -142.804, 52.32, 155.113]
  Call Extruder(0.00000)
  Set speed (18.0 mm/s)
  Call Extruder(4.37003)
  MoveL 10347 to (525.84, 523.95, 188) mm, rotated rx -180 ry 0 rz 160 deg; joints [8.724, 54.778, -8.768, -142.703, 52.477, 155.111]
  Set speed (18.0 mm/s)
  Call Extruder(8.89047)
  MoveL 10348 to (524.84, 524.98, 188) mm, rotated rx 180 ry 0 rz 160 deg; joints [8.864, 54.618, -8.474, -142.605, 52.643, 155.117]
  Set speed (18.0 mm/s)
  Call Extruder(11.20774)
  MoveL 10349 to (524.31, 525.5, 188) mm, rotated rx 180 ry 0 rz 160 deg; joints [8.935, 54.534, -8.319, -142.557, 52.73, 155.122]
  Set speed (18.0 mm/s)
  Call Extruder(13.43925)
  MoveL 10350 to (523.79, 525.99, 188) mm, rotated rx -180 ry 0 rz 160 deg; joints [9.002, 54.451, -8.165, -142.514, 52.814, 155.13]
  Call Extruder(16.27294)
  MoveL 10351 to (523.12, 526.59, 188) mm, rotated rx -180 ry 0 rz 160 deg; joints [9.086, 54.342, -7.965, -142.461, 52.922, 155.143]
  Set speed (18.0 mm/s)
  Call Extruder(21.22586)
  MoveL 10352 to (521.91, 527.6, 188) mm, rotated rx -180 ry 0 rz 160 deg; joints [9.228, 54.146, -7.601, -142.375, 53.114, 155.172]
  Set speed (18.0 mm/s)
  Call Extruder(25.41954)
  MoveL 10353 to (520.84, 528.41, 188) mm, rotated rx 180 ry 0 rz 160 deg; joints [9.345, 53.973, -7.282, -142.31, 53.279, 155.205]
  Set speed (18.0 mm/s)
  Call Extruder(29.47161)
  MoveL 10354 to (519.79, 529.15, 188) mm, rotated rx 180 ry 0 rz 160 deg; joints [9.454, 53.8, -6.962, -142.253, 53.441, 155.243]
  Set speed (18.0 mm/s)
  Call Extruder(31.62668)
  MoveL 10355 to (519.22, 529.53, 188) mm, rotated rx 180 ry 0 rz 160 deg; joints [9.511, 53.705, -6.789, -142.225, 53.527, 155.265]
  Call Extruder(36.00623)
  MoveL 10356 to (518.03, 530.27, 188) mm, rotated rx -180 ry 0 rz 160 deg; joints [9.622, 53.51, -6.428, -142.174, 53.704, 155.317]
  Call Extruder(38.52177)
  MoveL 10357 to (517.34, 530.67, 188) mm, rotated rx 180 ry 0 rz 160 deg; joints [9.684, 53.396, -6.217, -142.147, 53.807, 155.349]
  Set speed (18.0 mm/s)
  Call Extruder(40.57185)
  MoveL 10358 to (516.77, 530.99, 188) mm, rotated rx 180 ry 0 rz 160 deg; joints [9.734, 53.301, -6.042, -142.128, 53.89, 155.377]
  Set speed (18.0 mm/s)
  Call Extruder(42.88423)
  MoveL 10359 to (516.12, 531.33, 188) mm, rotated rx -180 ry 0 rz 160 deg; joints [9.788, 53.192, -5.842, -142.108, 53.985, 155.41]
  Call Extruder(47.35513)
  MoveL 10360 to (514.84, 531.96, 188) mm, rotated rx 180 ry 0 rz 160 deg; joints [9.889, 52.979, -5.449, -142.073, 54.169, 155.48]
  Call Extruder(51.88185)
  MoveL 10361 to (513.52, 532.54, 188) mm, rotated rx 180 ry 0 rz 160 deg; joints [9.987, 52.759, -5.043, -142.047, 54.356, 155.557]
  Set speed (18.0 mm/s)
  Call Extruder(56.39468)
  MoveL 10362 to (512.18, 533.06, 188) mm, rotated rx -180 ry 0 rz 160 deg; joints [10.078, 52.534, -4.629, -142.028, 54.543, 155.641]
  Set speed (18.0 mm/s)
  Call Extruder(60.89706)
  MoveL 10363 to (510.83, 533.53, 188) mm, rotated rx -180 ry 0 rz 160 deg; joints [10.164, 52.306, -4.208, -142.016, 54.73, 155.73]
  Set speed (17.9 mm/s)
  Call Extruder(62.64407)
  MoveL 10364 to (510.3, 533.7, 188) mm, rotated rx -180 ry 0 rz 160 deg; joints [10.195, 52.216, -4.044, -142.013, 54.802, 155.767]
  Set speed (18.0 mm/s)
  Call Extruder(65.81536)
  MoveL 10365 to (509.33, 533.98, 188) mm, rotated rx 180 ry 0 rz 160 deg; joints [10.25, 52.053, -3.742, -142.012, 54.934, 155.835]
  Set speed (18.0 mm/s)
  Call Extruder(69.93480)
  MoveL 10366 to (508.06, 534.3, 188) mm, rotated rx 180 ry 0 rz 160 deg; joints [10.317, 51.837, -3.345, -142.015, 55.104, 155.929]
  Set speed (18.0 mm/s)
  Call Extruder(74.63193)
  MoveL 10367 to (506.59, 534.61, 188) mm, rotated rx -180 ry 0 rz 160 deg; joints [10.388, 51.589, -2.888, -142.026, 55.297, 156.04]
  Call Extruder(79.20562)
  MoveL 10368 to (505.16, 534.85, 188) mm, rotated rx 180 ry 0 rz 160 deg; joints [10.45, 51.344, -2.437, -142.045, 55.484, 156.155]
  Set speed (18.0 mm/s)
  Call Extruder(83.55672)
  MoveL 10369 to (503.78, 535.03, 188) mm, rotated rx 180 ry 0 rz 160 deg; joints [10.502, 51.109, -2.005, -142.07, 55.661, 156.269]
  Set speed (18.0 mm/s)
  Call Extruder(88.21857)
  MoveL 10370 to (502.3, 535.16, 188) mm, rotated rx 180 ry 0 rz 160 deg; joints [10.551, 50.855, -1.539, -142.104, 55.848, 156.396]
  Call Extruder(92.79840)
  MoveL 10371 to (500.85, 535.22, 188) mm, rotated rx -180 ry 0 rz 160 deg; joints [10.593, 50.605, -1.079, -142.145, 56.03, 156.526]
  Set speed (10.0 mm/s)
  MoveL 10372 to (500.85, 535.22, 192) mm, rotated rx 180 ry 0 rz 160 deg; joints [10.593, 50.087, -1.048, -141.942, 55.647, 156.164]
  Set speed (120.0 mm/s)
  MoveL 10373 to (499.43, 535.1, 192) mm, rotated rx 180 ry 0 rz 160 deg; joints [10.61, 49.838, -0.593, -142.01, 55.816, 156.307]
  Set speed (18.0 mm/s)
  Call Extruder(97.35656)
  MoveL 10374 to (497.98, 535.04, 192) mm, rotated rx 180 ry 0 rz 160 deg; joints [10.637, 49.585, -0.132, -142.067, 55.991, 156.445]
  Set speed (18.0 mm/s)
  Call Extruder(101.87764)
  MoveL 10375 to (496.55, 534.93, 192) mm, rotated rx -180 ry 0 rz 160 deg; joints [10.656, 49.335, 0.325, -142.13, 56.161, 156.586]
  Set speed (18.0 mm/s)
  Call Extruder(106.32100)
  MoveL 10376 to (495.14, 534.76, 192) mm, rotated rx 180 ry 0 rz 160 deg; joints [10.668, 49.089, 0.774, -142.2, 56.326, 156.728]
  Set speed (18.0 mm/s)
  Call Extruder(110.78870)
  MoveL 10377 to (493.73, 534.54, 192) mm, rotated rx 180 ry 0 rz 160 deg; joints [10.673, 48.842, 1.224, -142.277, 56.488, 156.874]
  Set speed (18.0 mm/s)
  Call Extruder(115.43631)
  MoveL 10378 to (492.28, 534.24, 192) mm, rotated rx -180 ry 0 rz 160 deg; joints [10.67, 48.585, 1.69, -142.365, 56.654, 157.03]
  Set speed (18.0 mm/s)
  Call Extruder(119.75004)
  MoveL 10379 to (490.95, 533.91, 192) mm, rotated rx 180 ry 0 rz 160 deg; joints [10.661, 48.349, 2.12, -142.453, 56.803, 157.177]
  Set speed (18.0 mm/s)
  Call Extruder(124.42971)
  MoveL 10380 to (489.51, 533.5, 192) mm, rotated rx 180 ry 0 rz 160 deg; joints [10.642, 48.095, 2.582, -142.556, 56.961, 157.339]
  Call Extruder(128.76362)
  MoveL 10381 to (488.2, 533.06, 192) mm, rotated rx 180 ry 0 rz 160 deg; joints [10.618, 47.862, 3.007, -142.658, 57.104, 157.492]
  Set speed (18.0 mm/s)
  Call Extruder(133.39664)
  MoveL 10382 to (486.82, 532.53, 192) mm, rotated rx 180 ry 0 rz 160 deg; joints [10.584, 47.615, 3.455, -142.774, 57.251, 157.658]
  Set speed (18.0 mm/s)
  Call Extruder(135.62982)
  MoveL 10383 to (486.17, 532.26, 192) mm, rotated rx 180 ry 0 rz 160 deg; joints [10.565, 47.497, 3.669, -142.833, 57.321, 157.738]
  Set speed (18.0 mm/s)
  Call Extruder(140.16690)
  MoveL 10384 to (484.85, 531.66, 192) mm, rotated rx 180 ry 0 rz 160 deg; joints [10.52, 47.26, 4.1, -142.956, 57.458, 157.903]
  Set speed (18.0 mm/s)
  Call Extruder(143.10730)
  MoveL 10385 to (484.01, 531.25, 192) mm, rotated rx -180 ry 0 rz 160 deg; joints [10.487, 47.108, 4.375, -143.04, 57.544, 158.011]
  Set speed (18.0 mm/s)
  Call Extruder(146.80007)
  MoveL 10386 to (482.97, 530.69, 192) mm, rotated rx 180 ry 0 rz 160 deg; joints [10.441, 46.92, 4.716, -143.15, 57.649, 158.147]
  Set speed (18.0 mm/s)
  Call Extruder(151.29992)
  MoveL 10387 to (481.73, 529.97, 192) mm, rotated rx 180 ry 0 rz 160 deg; joints [10.377, 46.694, 5.126, -143.288, 57.773, 158.314]
  Set speed (18.0 mm/s)
  Call Extruder(155.12940)
  MoveL 10388 to (480.7, 529.32, 192) mm, rotated rx -180 ry 0 rz 160 deg; joints [10.318, 46.505, 5.469, -143.412, 57.875, 158.458]
  Set speed (18.0 mm/s)
  Call Extruder(158.05986)
  MoveL 10389 to (479.93, 528.79, 192) mm, rotated rx -180 ry 0 rz 160 deg; joints [10.268, 46.363, 5.726, -143.51, 57.949, 158.568]
  Set speed (18.0 mm/s)
  Call Extruder(160.25034)
  MoveL 10390 to (479.36, 528.39, 192) mm, rotated rx 180 ry 0 rz 160 deg; joints [10.229, 46.258, 5.917, -143.584, 58.003, 158.65]
  Set speed (18.0 mm/s)
  Call Extruder(164.71066)
  MoveL 10391 to (478.22, 527.53, 192) mm, rotated rx 180 ry 0 rz 160 deg; joints [10.144, 46.048, 6.297, -143.741, 58.109, 158.819]
  Set speed (18.0 mm/s)
  Call Extruder(167.16515)
  MoveL 10392 to (477.62, 527.04, 192) mm, rotated rx 180 ry 0 rz 160 deg; joints [10.094, 45.935, 6.502, -143.829, 58.165, 158.911]
  Set speed (18.0 mm/s)
  Call Extruder(169.33685)
  MoveL 10393 to (477.09, 526.59, 192) mm, rotated rx -180 ry 0 rz 160 deg; joints [10.048, 45.836, 6.681, -143.909, 58.214, 158.994]
  Set speed (18.0 mm/s)
  Call Extruder(173.88179)
  MoveL 10394 to (476.01, 525.62, 192) mm, rotated rx 180 ry 0 rz 160 deg; joints [9.946, 45.633, 7.047, -144.08, 58.31, 159.165]
  Set speed (18.0 mm/s)
  Call Extruder(176.09735)
  MoveL 10395 to (475.5, 525.13, 192) mm, rotated rx 180 ry 0 rz 160 deg; joints [9.894, 45.537, 7.221, -144.165, 58.354, 159.249]
  Set speed (18.0 mm/s)
  Call Extruder(180.15559)
  MoveL 10396 to (474.58, 524.22, 192) mm, rotated rx 180 ry 0 rz 160 deg; joints [9.795, 45.364, 7.534, -144.325, 58.433, 159.402]
  Set speed (18.0 mm/s)
  Call Extruder(185.03642)
  MoveL 10397 to (473.54, 523.06, 192) mm, rotated rx 180 ry 0 rz 160 deg; joints [9.666, 45.163, 7.896, -144.523, 58.519, 159.586]
  Set speed (18.0 mm/s)
  Call Extruder(187.33879)
  MoveL 10398 to (473.06, 522.5, 192) mm, rotated rx 180 ry 0 rz 160 deg; joints [9.604, 45.072, 8.062, -144.619, 58.558, 159.673]
  Call Extruder(189.61017)
  MoveL 10399 to (472.6, 521.94, 192) mm, rotated rx 180 ry 0 rz 160 deg; joints [9.54, 44.983, 8.222, -144.714, 58.594, 159.758]
  Call Extruder(191.83254)
  MoveL 10400 to (472.17, 521.39, 192) mm, rotated rx 180 ry 0 rz 160 deg; joints [9.476, 44.898, 8.376, -144.809, 58.628, 159.841]
  Call Extruder(196.34474)
  MoveL 10401 to (471.31, 520.23, 192) mm, rotated rx -180 ry 0 rz 160 deg; joints [9.341, 44.73, 8.678, -145.004, 58.692, 160.008]
  Set speed (18.0 mm/s)
  Call Extruder(200.76980)
  MoveL 10402 to (470.53, 519.06, 192) mm, rotated rx 180 ry 0 rz 160 deg; joints [9.203, 44.574, 8.96, -145.2, 58.748, 160.172]
  Call Extruder(203.18633)
  MoveL 10403 to (470.11, 518.41, 192) mm, rotated rx -180 ry 0 rz 160 deg; joints [9.125, 44.491, 9.11, -145.308, 58.776, 160.26]
  Call Extruder(207.67740)
  MoveL 10404 to (469.39, 517.17, 192) mm, rotated rx -180 ry 0 rz 160 deg; joints [8.976, 44.344, 9.375, -145.513, 58.823, 160.424]
  Call Extruder(210.13719)
  MoveL 10405 to (469.01, 516.48, 192) mm, rotated rx 180 ry 0 rz 160 deg; joints [8.892, 44.267, 9.514, -145.627, 58.846, 160.513]
  Set speed (18.0 mm/s)
  Call Extruder(214.30163)
  MoveL 10406 to (468.41, 515.3, 192) mm, rotated rx -180 ry 0 rz 160 deg; joints [8.746, 44.142, 9.739, -145.822, 58.88, 160.662]
  Set speed (18.0 mm/s)
  Call Extruder(218.80554)
  MoveL 10407 to (467.81, 513.99, 192) mm, rotated rx 180 ry 0 rz 160 deg; joints [8.583, 44.015, 9.967, -146.036, 58.911, 160.821]
  Call Extruder(223.44533)
  MoveL 10408 to (467.25, 512.62, 192) mm, rotated rx -180 ry 0 rz 160 deg; joints [8.41, 43.894, 10.186, -146.259, 58.935, 160.983]
  Set speed (18.0 mm/s)
  Call Extruder(228.05066)
  MoveL 10409 to (466.75, 511.24, 192) mm, rotated rx -180 ry 0 rz 160 deg; joints [8.234, 43.783, 10.386, -146.483, 58.952, 161.141]
  Call Extruder(232.32744)
  MoveL 10410 to (466.34, 509.94, 192) mm, rotated rx 180 ry 0 rz 160 deg; joints [8.066, 43.688, 10.556, -146.694, 58.961, 161.285]
  Call Extruder(237.56396)
  MoveL 10411 to (465.9, 508.33, 192) mm, rotated rx 180 ry 0 rz 160 deg; joints [7.857, 43.583, 10.745, -146.953, 58.964, 161.458]
  Set speed (18.0 mm/s)
  Call Extruder(242.05523)
  MoveL 10412 to (465.59, 506.94, 192) mm, rotated rx 180 ry 0 rz 160 deg; joints [7.673, 43.504, 10.887, -147.177, 58.959, 161.602]
  Set speed (18.0 mm/s)
  Call Extruder(245.98205)
  MoveL 10413 to (465.37, 505.71, 192) mm, rotated rx -180 ry 0 rz 160 deg; joints [7.51, 43.443, 10.997, -147.373, 58.949, 161.726]
  Set speed (18.0 mm/s)
  Call Extruder(250.49645)
  MoveL 10414 to (465.16, 504.28, 192) mm, rotated rx -180 ry 0 rz 160 deg; joints [7.32, 43.381, 11.108, -147.6, 58.931, 161.866]
  Set speed (18.0 mm/s)
  Call Extruder(254.99004)
  MoveL 10415 to (465.02, 502.86, 192) mm, rotated rx -180 ry 0 rz 160 deg; joints [7.129, 43.33, 11.2, -147.826, 58.907, 162.001]
  Set speed (18.0 mm/s)
  Call Extruder(259.35006)
  MoveL 10416 to (464.93, 501.47, 192) mm, rotated rx 180 ry 0 rz 160 deg; joints [6.941, 43.289, 11.273, -148.044, 58.876, 162.129]
  Call Extruder(263.96956)
  MoveL 10417 to (464.9, 500, 192) mm, rotated rx 180 ry 0 rz 160 deg; joints [6.741, 43.257, 11.332, -148.275, 58.837, 162.26]
  Call Extruder(267.86069)
  MoveL 10418 to (464.92, 498.76, 192) mm, rotated rx 180 ry 0 rz 160 deg; joints [6.571, 43.237, 11.367, -148.469, 58.799, 162.368]
  Call Extruder(271.97715)
  MoveL 10419 to (464.99, 497.45, 192) mm, rotated rx 180 ry 0 rz 160 deg; joints [6.391, 43.225, 11.389, -148.673, 58.753, 162.478]
  Set speed (18.0 mm/s)
  Call Extruder(276.08991)
  MoveL 10420 to (465.11, 496.14, 192) mm, rotated rx 180 ry 0 rz 160 deg; joints [6.211, 43.221, 11.396, -148.875, 58.701, 162.584]
  Set speed (18.0 mm/s)
  Call Extruder(280.13914)
  MoveL 10421 to (465.28, 494.86, 192) mm, rotated rx 180 ry 0 rz 160 deg; joints [6.034, 43.225, 11.388, -149.072, 58.645, 162.685]
  Set speed (18.0 mm/s)
  Call Extruder(284.27384)
  MoveL 10422 to (465.5, 493.56, 192) mm, rotated rx -180 ry 0 rz 160 deg; joints [5.853, 43.238, 11.365, -149.271, 58.583, 162.784]
  Set speed (18.0 mm/s)
  Call Extruder(288.23847)
  MoveL 10423 to (465.75, 492.32, 192) mm, rotated rx -180 ry 0 rz 160 deg; joints [5.68, 43.259, 11.328, -149.46, 58.518, 162.875]
  Set speed (18.0 mm/s)
  Call Extruder(292.28997)
  MoveL 10424 to (466.05, 491.07, 192) mm, rotated rx 180 ry 0 rz 160 deg; joints [5.504, 43.287, 11.277, -149.65, 58.447, 162.965]
  Set speed (18.0 mm/s)
  Call Extruder(296.33883)
  MoveL 10425 to (466.41, 489.83, 192) mm, rotated rx -180 ry 0 rz 160 deg; joints [5.33, 43.325, 11.209, -149.836, 58.37, 163.049]
  Call Extruder(300.35219)
  MoveL 10426 to (466.8, 488.61, 192) mm, rotated rx -180 ry 0 rz 160 deg; joints [5.159, 43.369, 11.129, -150.018, 58.289, 163.13]
  Set speed (18.0 mm/s)
  Call Extruder(304.39378)
  MoveL 10427 to (467.24, 487.4, 192) mm, rotated rx -180 ry 0 rz 160 deg; joints [4.988, 43.422, 11.034, -150.197, 58.203, 163.206]
  Set speed (18.0 mm/s)
  Call Extruder(306.91450)
  MoveL 10428 to (467.55, 486.65, 192) mm, rotated rx -180 ry 0 rz 160 deg; joints [4.883, 43.46, 10.966, -150.306, 58.147, 163.251]
  Set speed (18.0 mm/s)
  Call Extruder(307.79235)
  MoveL 10429 to (467.64, 486.39, 192) mm, rotated rx -180 ry 0 rz 160 deg; joints [4.846, 43.472, 10.944, -150.345, 58.128, 163.267]
  Set speed (18.0 mm/s)
  Call Extruder(312.59937)
  MoveL 10430 to (468.27, 484.99, 192) mm, rotated rx -180 ry 0 rz 160 deg; joints [4.649, 43.553, 10.799, -150.548, 58.015, 163.348]
  Set speed (18.0 mm/s)
  Call Extruder(316.57258)
  MoveL 10431 to (468.83, 483.86, 192) mm, rotated rx 180 ry 0 rz 160 deg; joints [4.488, 43.628, 10.663, -150.711, 57.916, 163.409]
  Set speed (18.0 mm/s)
  Call Extruder(320.60891)
  MoveL 10432 to (469.44, 482.73, 192) mm, rotated rx 180 ry 0 rz 160 deg; joints [4.327, 43.712, 10.513, -150.872, 57.812, 163.467]
  Set speed (18.0 mm/s)
  Call Extruder(324.57644)
  MoveL 10433 to (470.09, 481.64, 192) mm, rotated rx -180 ry 0 rz 160 deg; joints [4.173, 43.802, 10.352, -151.025, 57.706, 163.52]
  Call Extruder(328.69172)
  MoveL 10434 to (470.79, 480.53, 192) mm, rotated rx 180 ry 0 rz 160 deg; joints [4.016, 43.902, 10.171, -151.179, 57.591, 163.569]
  Set speed (18.0 mm/s)
  Call Extruder(332.69046)
  MoveL 10435 to (471.52, 479.49, 192) mm, rotated rx -180 ry 0 rz 160 deg; joints [3.867, 44.007, 9.982, -151.323, 57.475, 163.612]
  Set speed (18.0 mm/s)
  Call Extruder(336.72407)
  MoveL 10436 to (472.29, 478.46, 192) mm, rotated rx -180 ry 0 rz 160 deg; joints [3.72, 44.119, 9.779, -151.462, 57.355, 163.651]
  Set speed (18.0 mm/s)
  Call Extruder(340.86598)
  MoveL 10437 to (473.12, 477.43, 192) mm, rotated rx -180 ry 0 rz 160 deg; joints [3.574, 44.242, 9.558, -151.598, 57.227, 163.685]
  Call Extruder(344.98950)
  MoveL 10438 to (473.99, 476.44, 192) mm, rotated rx 180 ry 0 rz 160 deg; joints [3.433, 44.371, 9.325, -151.727, 57.096, 163.714]
  Set speed (18.0 mm/s)
  Call Extruder(349.13062)
  MoveL 10439 to (474.89, 475.48, 192) mm, rotated rx 180 ry 0 rz 160 deg; joints [3.297, 44.508, 9.079, -151.85, 56.961, 163.737]
  Set speed (18.0 mm/s)
  Call Extruder(352.99932)
  MoveL 10440 to (475.77, 474.61, 192) mm, rotated rx 180 ry 0 rz 160 deg; joints [3.174, 44.642, 8.838, -151.958, 56.832, 163.753]
  Set speed (18.0 mm/s)
  Call Extruder(357.07701)
  MoveL 10441 to (476.72, 473.73, 192) mm, rotated rx 180 ry 0 rz 160 deg; joints [3.048, 44.789, 8.572, -152.066, 56.692, 163.766]
  Set speed (18.0 mm/s)
  Call Extruder(361.23438)
  MoveL 10442 to (477.73, 472.87, 192) mm, rotated rx 180 ry 0 rz 160 deg; joints [2.926, 44.945, 8.29, -152.167, 56.547, 163.773]
  Set speed (18.0 mm/s)
  Call Extruder(365.18705)
  MoveL 10443 to (478.72, 472.09, 192) mm, rotated rx 180 ry 0 rz 160 deg; joints [2.815, 45.099, 8.011, -152.257, 56.406, 163.774]
  Set speed (17.9 mm/s)
  Call Extruder(367.34066)
  MoveL 10444 to (479.26, 471.67, 192) mm, rotated rx 180 ry 0 rz 160 deg; joints [2.756, 45.185, 7.857, -152.304, 56.328, 163.773]
  Set speed (17.9 mm/s)
  Call Extruder(369.18925)
  MoveL 10445 to (479.75, 471.34, 192) mm, rotated rx -180 ry 0 rz 160 deg; joints [2.708, 45.261, 7.72, -152.34, 56.261, 163.77]
  Set speed (18.0 mm/s)
  Call Extruder(373.40821)
  MoveL 10446 to (480.86, 470.58, 192) mm, rotated rx 180 ry 0 rz 160 deg; joints [2.601, 45.437, 7.401, -152.42, 56.105, 163.759]
  Set speed (18.0 mm/s)
  Call Extruder(377.50703)
  MoveL 10447 to (481.97, 469.89, 192) mm, rotated rx 180 ry 0 rz 160 deg; joints [2.502, 45.614, 7.082, -152.49, 55.951, 163.743]
  Set speed (18.0 mm/s)
  Call Extruder(381.55395)
  MoveL 10448 to (483.09, 469.24, 192) mm, rotated rx -180 ry 0 rz 160 deg; joints [2.411, 45.793, 6.758, -152.55, 55.796, 163.722]
  Call Extruder(385.47146)
  MoveL 10449 to (484.19, 468.66, 192) mm, rotated rx 180 ry 0 rz 160 deg; joints [2.328, 45.971, 6.435, -152.601, 55.645, 163.696]
  Call Extruder(389.61302)
  MoveL 10450 to (485.38, 468.09, 192) mm, rotated rx 180 ry 0 rz 160 deg; joints [2.246, 46.164, 6.086, -152.647, 55.483, 163.663]
  Call Extruder(393.71486)
  MoveL 10451 to (486.58, 467.57, 192) mm, rotated rx 180 ry 0 rz 160 deg; joints [2.171, 46.36, 5.732, -152.684, 55.321, 163.624]
  Set speed (18.0 mm/s)
  Call Extruder(397.59277)
  MoveL 10452 to (487.73, 467.11, 192) mm, rotated rx 180 ry 0 rz 160 deg; joints [2.106, 46.548, 5.39, -152.711, 55.167, 163.581]
  Set speed (18.0 mm/s)
  Call Extruder(401.79166)
  MoveL 10453 to (489, 466.67, 192) mm, rotated rx 180 ry 0 rz 160 deg; joints [2.042, 46.757, 5.013, -152.732, 54.998, 163.53]
  Set speed (18.0 mm/s)
  Call Extruder(405.72598)
  MoveL 10454 to (490.19, 466.3, 192) mm, rotated rx -180 ry 0 rz 160 deg; joints [1.988, 46.955, 4.653, -152.743, 54.84, 163.476]
  Set speed (18.0 mm/s)
  Call Extruder(409.92417)
  MoveL 10455 to (491.49, 465.95, 192) mm, rotated rx 180 ry 0 rz 160 deg; joints [1.937, 47.17, 4.263, -152.747, 54.669, 163.412]
  Set speed (18.0 mm/s)
  Call Extruder(413.77383)
  MoveL 10456 to (492.68, 465.67, 192) mm, rotated rx -180 ry 0 rz 160 deg; joints [1.896, 47.37, 3.9, -152.742, 54.513, 163.349]
  Set speed (18.0 mm/s)
  Call Extruder(417.87307)
  MoveL 10457 to (493.96, 465.43, 192) mm, rotated rx -180 ry 0 rz 160 deg; joints [1.858, 47.585, 3.508, -152.729, 54.346, 163.275]
  Set speed (18.0 mm/s)
  Call Extruder(421.78129)
  MoveL 10458 to (495.19, 465.23, 192) mm, rotated rx -180 ry 0 rz 160 deg; joints [1.828, 47.793, 3.131, -152.708, 54.186, 163.2]
  Set speed (18.0 mm/s)
  Call Extruder(426.07958)
  MoveL 10459 to (496.56, 465.07, 192) mm, rotated rx 180 ry 0 rz 160 deg; joints [1.802, 48.024, 2.712, -152.677, 54.011, 163.111]
  Set speed (18.0 mm/s)
  Call Extruder(430.06103)
  MoveL 10460 to (497.82, 464.97, 192) mm, rotated rx 180 ry 0 rz 160 deg; joints [1.784, 48.239, 2.32, -152.639, 53.849, 163.024]
  Set speed (18.0 mm/s)
  Call Extruder(434.24260)
  MoveL 10461 to (499.15, 464.91, 192) mm, rotated rx 180 ry 0 rz 160 deg; joints [1.771, 48.468, 1.904, -152.591, 53.679, 162.926]
  Set speed (18.0 mm/s)
  Call Extruder(438.21718)
  MoveL 10462 to (500.42, 464.9, 192) mm, rotated rx 180 ry 0 rz 160 deg; joints [1.765, 48.686, 1.507, -152.537, 53.518, 162.828]
  Set speed (18.0 mm/s)
  Call Extruder(442.35492)
  MoveL 10463 to (501.74, 464.94, 192) mm, rotated rx -180 ry 0 rz 160 deg; joints [1.765, 48.915, 1.091, -152.473, 53.352, 162.72]
  Set speed (18.0 mm/s)
  Call Extruder(446.33834)
  MoveL 10464 to (503.01, 465.03, 192) mm, rotated rx -180 ry 0 rz 160 deg; joints [1.771, 49.135, 0.689, -152.403, 53.193, 162.611]
  Set speed (18.0 mm/s)
  Call Extruder(450.24671)
  MoveL 10465 to (504.25, 465.16, 192) mm, rotated rx 180 ry 0 rz 160 deg; joints [1.783, 49.352, 0.294, -152.327, 53.039, 162.499]
  Set speed (18.0 mm/s)
  Call Extruder(454.35338)
  MoveL 10466 to (505.54, 465.34, 192) mm, rotated rx 180 ry 0 rz 160 deg; joints [1.801, 49.579, -0.121, -152.24, 52.878, 162.377]
  Set speed (18.0 mm/s)
  Call Extruder(458.55312)
  MoveL 10467 to (506.86, 465.58, 192) mm, rotated rx 180 ry 0 rz 160 deg; joints [1.825, 49.812, -0.546, -152.143, 52.716, 162.247]
  Set speed (18.0 mm/s)
  Call Extruder(462.54318)
  MoveL 10468 to (508.1, 465.85, 192) mm, rotated rx -180 ry 0 rz 160 deg; joints [1.854, 50.033, -0.949, -152.043, 52.563, 162.119]
  Set speed (18.0 mm/s)
  Call Extruder(466.77999)
  MoveL 10469 to (509.41, 466.19, 192) mm, rotated rx -180 ry 0 rz 160 deg; joints [1.891, 50.267, -1.376, -151.929, 52.404, 161.978]
  Set speed (18.0 mm/s)
  Call Extruder(470.63805)
  MoveL 10470 to (510.59, 466.54, 192) mm, rotated rx -180 ry 0 rz 160 deg; joints [1.93, 50.479, -1.763, -151.819, 52.262, 161.845]
  Set speed (18.0 mm/s)
  Call Extruder(474.75141)
  MoveL 10471 to (511.84, 466.96, 192) mm, rotated rx 180 ry 0 rz 160 deg; joints [1.977, 50.703, -2.173, -151.694, 52.113, 161.699]
  Set speed (18.0 mm/s)
  Call Extruder(478.57964)
  MoveL 10472 to (512.98, 467.39, 192) mm, rotated rx 180 ry 0 rz 160 deg; joints [2.025, 50.911, -2.553, -151.572, 51.977, 161.559]
  Call Extruder(482.86880)
  MoveL 10473 to (514.24, 467.92, 192) mm, rotated rx 180 ry 0 rz 160 deg; joints [2.085, 51.142, -2.975, -151.429, 51.828, 161.399]
  Set speed (18.0 mm/s)
  Call Extruder(486.68821)
  MoveL 10474 to (515.35, 468.43, 192) mm, rotated rx -180 ry 0 rz 160 deg; joints [2.143, 51.345, -3.347, -151.295, 51.699, 161.253]
  Call Extruder(490.86785)
  MoveL 10475 to (516.53, 469.04, 192) mm, rotated rx 180 ry 0 rz 160 deg; joints [2.212, 51.565, -3.749, -151.142, 51.561, 161.089]
  Set speed (18.0 mm/s)
  Call Extruder(494.99615)
  MoveL 10476 to (517.68, 469.68, 192) mm, rotated rx -180 ry 0 rz 160 deg; joints [2.285, 51.779, -4.141, -150.985, 51.429, 160.924]
  Call Extruder(498.93388)
  MoveL 10477 to (518.75, 470.33, 192) mm, rotated rx -180 ry 0 rz 160 deg; joints [2.36, 51.98, -4.51, -150.83, 51.307, 160.763]
  Set speed (18.0 mm/s)
  Call Extruder(502.87116)
  MoveL 10478 to (519.8, 471.02, 192) mm, rotated rx -180 ry 0 rz 160 deg; joints [2.439, 52.179, -4.873, -150.67, 51.189, 160.6]
  Call Extruder(507.01275)
  MoveL 10479 to (520.88, 471.79, 192) mm, rotated rx 180 ry 0 rz 160 deg; joints [2.526, 52.383, -5.248, -150.496, 51.07, 160.426]
  Call Extruder(511.12821)
  MoveL 10480 to (521.92, 472.59, 192) mm, rotated rx 180 ry 0 rz 160 deg; joints [2.618, 52.583, -5.614, -150.319, 50.956, 160.251]
  Set speed (18.0 mm/s)
  Call Extruder(515.17963)
  MoveL 10481 to (522.92, 473.41, 192) mm, rotated rx 180 ry 0 rz 160 deg; joints [2.712, 52.775, -5.967, -150.14, 50.849, 160.076]
  Set speed (18.0 mm/s)
  Call Extruder(519.27583)
  MoveL 10482 to (523.89, 474.29, 192) mm, rotated rx -180 ry 0 rz 160 deg; joints [2.812, 52.965, -6.314, -149.954, 50.746, 159.898]
  Set speed (18.0 mm/s)
  Call Extruder(523.35127)
  MoveL 10483 to (524.82, 475.19, 192) mm, rotated rx -180 ry 0 rz 160 deg; joints [2.915, 53.148, -6.651, -149.766, 50.649, 159.719]
  Set speed (18.0 mm/s)
  Call Extruder(527.70102)
  MoveL 10484 to (525.79, 476.19, 192) mm, rotated rx -180 ry 0 rz 160 deg; joints [3.03, 53.339, -7.002, -149.561, 50.551, 159.527]
  Call Extruder(532.14238)
  MoveL 10485 to (526.73, 477.25, 192) mm, rotated rx -180 ry 0 rz 160 deg; joints [3.151, 53.527, -7.347, -149.348, 50.459, 159.329]
  Set speed (18.0 mm/s)
  Call Extruder(534.45387)
  MoveL 10486 to (527.2, 477.81, 192) mm, rotated rx -180 ry 0 rz 160 deg; joints [3.216, 53.623, -7.523, -149.236, 50.413, 159.226]
  Set speed (18.0 mm/s)
  Call Extruder(536.71196)
  MoveL 10487 to (527.65, 478.38, 192) mm, rotated rx 180 ry 0 rz 160 deg; joints [3.28, 53.714, -7.691, -149.126, 50.37, 159.126]
  Set speed (18.0 mm/s)
  Call Extruder(541.15491)
  MoveL 10488 to (528.5, 479.51, 192) mm, rotated rx 180 ry 0 rz 160 deg; joints [3.41, 53.889, -8.011, -148.906, 50.291, 158.928]
  Call Extruder(543.48330)
  MoveL 10489 to (528.92, 480.12, 192) mm, rotated rx 180 ry 0 rz 160 deg; joints [3.479, 53.977, -8.173, -148.79, 50.253, 158.824]
  Set speed (18.0 mm/s)
  Call Extruder(545.71452)
  MoveL 10490 to (529.32, 480.71, 192) mm, rotated rx -180 ry 0 rz 160 deg; joints [3.547, 54.06, -8.326, -148.678, 50.218, 158.725]
  Set speed (18.0 mm/s)
  Call Extruder(548.12219)
  MoveL 10491 to (529.74, 481.35, 192) mm, rotated rx -180 ry 0 rz 160 deg; joints [3.62, 54.147, -8.486, -148.557, 50.182, 158.618]
  Set speed (18.0 mm/s)
  Call Extruder(550.24330)
  MoveL 10492 to (530.09, 481.93, 192) mm, rotated rx -180 ry 0 rz 160 deg; joints [3.687, 54.222, -8.624, -148.449, 50.153, 158.524]
  Set speed (18.0 mm/s)
  Call Extruder(552.54110)
  MoveL 10493 to (530.46, 482.56, 192) mm, rotated rx -180 ry 0 rz 160 deg; joints [3.759, 54.301, -8.769, -148.333, 50.123, 158.423]
  Set speed (18.0 mm/s)
  Call Extruder(554.83331)
  MoveL 10494 to (530.82, 483.2, 192) mm, rotated rx -180 ry 0 rz 160 deg; joints [3.832, 54.378, -8.911, -148.216, 50.095, 158.322]
  Set speed (18.0 mm/s)
  Call Extruder(556.99960)
  MoveL 10495 to (531.14, 483.81, 192) mm, rotated rx 180 ry 0 rz 160 deg; joints [3.902, 54.449, -9.04, -148.105, 50.071, 158.227]
  Call Extruder(559.50474)
  MoveL 10496 to (531.5, 484.52, 192) mm, rotated rx -180 ry 0 rz 160 deg; joints [3.983, 54.528, -9.186, -147.977, 50.045, 158.117]
  Set speed (18.0 mm/s)
  Call Extruder(562.59633)
  MoveL 10497 to (531.92, 485.41, 192) mm, rotated rx -180 ry 0 rz 160 deg; joints [4.085, 54.622, -9.358, -147.819, 50.016, 157.984]
  Set speed (18.0 mm/s)
  Call Extruder(566.11789)
  MoveL 10498 to (532.37, 486.44, 192) mm, rotated rx 180 ry 0 rz 160 deg; joints [4.203, 54.723, -9.544, -147.638, 49.989, 157.833]
  Set speed (18.0 mm/s)
  Call Extruder(568.35976)
  MoveL 10499 to (532.64, 487.1, 192) mm, rotated rx -180 ry 0 rz 160 deg; joints [4.279, 54.785, -9.659, -147.523, 49.973, 157.737]
  Set speed (18.0 mm/s)
  Call Extruder(572.96907)
  MoveL 10500 to (533.15, 488.48, 192) mm, rotated rx -180 ry 0 rz 160 deg; joints [4.437, 54.905, -9.879, -147.286, 49.949, 157.544]
  Set speed (18.0 mm/s)
  Call Extruder(577.28609)
  MoveL 10501 to (533.58, 489.78, 192) mm, rotated rx 180 ry 0 rz 160 deg; joints [4.587, 55.008, -10.069, -147.065, 49.933, 157.366]
  Set speed (18.0 mm/s)
  Call Extruder(581.67221)
  MoveL 10502 to (533.96, 491.13, 192) mm, rotated rx -180 ry 0 rz 160 deg; joints [4.742, 55.104, -10.246, -146.842, 49.926, 157.188]
  Set speed (18.0 mm/s)
  Call Extruder(586.25854)
  MoveL 10503 to (534.3, 492.55, 192) mm, rotated rx 180 ry 0 rz 160 deg; joints [4.906, 55.194, -10.412, -146.609, 49.926, 157.006]
  Set speed (18.0 mm/s)
  Call Extruder(590.83332)
  MoveL 10504 to (534.58, 493.98, 192) mm, rotated rx 180 ry 0 rz 160 deg; joints [5.071, 55.273, -10.558, -146.38, 49.935, 156.83]
  Call Extruder(595.33416)
  MoveL 10505 to (534.8, 495.4, 192) mm, rotated rx -180 ry 0 rz 160 deg; joints [5.236, 55.341, -10.682, -146.156, 49.953, 156.662]
  Set speed (18.0 mm/s)
  Call Extruder(599.93983)
  MoveL 10506 to (534.96, 496.86, 192) mm, rotated rx 180 ry 0 rz 160 deg; joints [5.405, 55.4, -10.791, -145.929, 49.979, 156.495]
  Call Extruder(604.34931)
  MoveL 10507 to (535.06, 498.27, 192) mm, rotated rx 180 ry 0 rz 160 deg; joints [5.569, 55.446, -10.875, -145.716, 50.012, 156.341]
  Set speed (18.0 mm/s)
  Call Extruder(608.83917)
  MoveL 10508 to (535.1, 499.7, 192) mm, rotated rx -180 ry 0 rz 160 deg; joints [5.736, 55.482, -10.941, -145.502, 50.055, 156.191]
  Set speed (18.0 mm/s)
  Call Extruder(613.23577)
  MoveL 10509 to (535.08, 501.1, 192) mm, rotated rx -180 ry 0 rz 160 deg; joints [5.9, 55.506, -10.987, -145.296, 50.104, 156.05]
  Set speed (18.0 mm/s)
  Call Extruder(617.85349)
  MoveL 10510 to (535.01, 502.57, 192) mm, rotated rx 180 ry 0 rz 160 deg; joints [6.073, 55.522, -11.016, -145.084, 50.164, 155.908]
  Call Extruder(622.27145)
  MoveL 10511 to (534.87, 503.97, 192) mm, rotated rx 180 ry 0 rz 160 deg; joints [6.239, 55.526, -11.023, -144.885, 50.229, 155.779]
  Call Extruder(626.95087)
  MoveL 10512 to (534.67, 505.45, 192) mm, rotated rx 180 ry 0 rz 160 deg; joints [6.414, 55.519, -11.009, -144.68, 50.306, 155.651]
  Set speed (18.0 mm/s)
  Call Extruder(631.26482)
  MoveL 10513 to (534.43, 506.81, 192) mm, rotated rx 180 ry 0 rz 160 deg; joints [6.576, 55.502, -10.979, -144.496, 50.384, 155.54]
  Call Extruder(635.90571)
  MoveL 10514 to (534.12, 508.25, 192) mm, rotated rx -180 ry 0 rz 160 deg; joints [6.749, 55.472, -10.924, -144.303, 50.477, 155.428]
  Set speed (18.0 mm/s)
  Call Extruder(640.39223)
  MoveL 10515 to (533.75, 509.64, 192) mm, rotated rx 180 ry 0 rz 160 deg; joints [6.916, 55.433, -10.852, -144.122, 50.573, 155.328]
  Set speed (18.0 mm/s)
  Call Extruder(644.88131)
  MoveL 10516 to (533.33, 511, 192) mm, rotated rx 180 ry 0 rz 160 deg; joints [7.082, 55.384, -10.761, -143.947, 50.676, 155.236]
  Set speed (18.0 mm/s)
  Call Extruder(649.28705)
  MoveL 10517 to (532.87, 512.33, 192) mm, rotated rx -180 ry 0 rz 160 deg; joints [7.244, 55.325, -10.653, -143.782, 50.784, 155.154]
  Set speed (18.0 mm/s)
  Call Extruder(653.77101)
  MoveL 10518 to (532.34, 513.66, 192) mm, rotated rx -180 ry 0 rz 160 deg; joints [7.407, 55.256, -10.525, -143.619, 50.899, 155.078]
  Set speed (18.0 mm/s)
  Call Extruder(659.21723)
  MoveL 10519 to (531.62, 515.24, 192) mm, rotated rx -180 ry 0 rz 160 deg; joints [7.603, 55.157, -10.343, -143.43, 51.049, 154.997]
  Set speed (18.0 mm/s)
  Call Extruder(662.73292)
  MoveL 10520 to (531.12, 516.24, 192) mm, rotated rx 180 ry 0 rz 160 deg; joints [7.728, 55.085, -10.211, -143.314, 51.15, 154.952]
  Set speed (18.0 mm/s)
  Call Extruder(667.37278)
  MoveL 10521 to (530.41, 517.53, 192) mm, rotated rx 180 ry 0 rz 160 deg; joints [7.892, 54.981, -10.02, -143.166, 51.289, 154.9]
  Call Extruder(669.59339)
  MoveL 10522 to (530.05, 518.14, 192) mm, rotated rx -180 ry 0 rz 160 deg; joints [7.969, 54.928, -9.922, -143.097, 51.358, 154.878]
  Set speed (18.0 mm/s)
  Call Extruder(671.80976)
  MoveL 10523 to (529.68, 518.75, 192) mm, rotated rx 180 ry 0 rz 160 deg; joints [8.046, 54.872, -9.82, -143.031, 51.428, 154.859]
  Set speed (18.0 mm/s)
  Call Extruder(674.70519)
  MoveL 10524 to (529.17, 519.52, 192) mm, rotated rx -180 ry 0 rz 160 deg; joints [8.145, 54.797, -9.68, -142.947, 51.521, 154.836]
  Set speed (18.0 mm/s)
  Call Extruder(678.54439)
  MoveL 10525 to (528.47, 520.52, 192) mm, rotated rx -180 ry 0 rz 160 deg; joints [8.275, 54.689, -9.483, -142.84, 51.648, 154.812]
  Set speed (18.0 mm/s)
  Call Extruder(680.91783)
  MoveL 10526 to (528.02, 521.14, 192) mm, rotated rx 180 ry 0 rz 160 deg; joints [8.354, 54.621, -9.356, -142.776, 51.728, 154.8]
  Set speed (18.0 mm/s)
  Call Extruder(684.42566)
  MoveL 10527 to (527.34, 522.02, 192) mm, rotated rx 180 ry 0 rz 160 deg; joints [8.47, 54.514, -9.16, -142.685, 51.848, 154.787]
  Set speed (18.0 mm/s)
  Call Extruder(689.85023)
  MoveL 10528 to (526.22, 523.34, 192) mm, rotated rx 180 ry 0 rz 160 deg; joints [8.645, 54.337, -8.835, -142.554, 52.041, 154.777]
  Set speed (18.0 mm/s)
  Call Extruder(693.84428)
  MoveL 10529 to (525.35, 524.28, 192) mm, rotated rx 180 ry 0 rz 160 deg; joints [8.771, 54.2, -8.584, -142.464, 52.185, 154.777]
  Call Extruder(696.56105)
  MoveL 10530 to (524.75, 524.89, 192) mm, rotated rx 180 ry 0 rz 160 deg; joints [8.855, 54.103, -8.405, -142.407, 52.286, 154.781]
  Set speed (18.0 mm/s)
  Call Extruder(698.90496)
  MoveL 10531 to (524.21, 525.41, 192) mm, rotated rx -180 ry 0 rz 160 deg; joints [8.926, 54.017, -8.247, -142.359, 52.373, 154.786]
  Set speed (18.0 mm/s)
  Call Extruder(703.30695)
  MoveL 10532 to (523.18, 526.36, 192) mm, rotated rx -180 ry 0 rz 160 deg; joints [9.058, 53.85, -7.94, -142.275, 52.54, 154.803]
  Set speed (18.0 mm/s)
  Call Extruder(705.57645)
  MoveL 10533 to (522.63, 526.83, 192) mm, rotated rx -180 ry 0 rz 160 deg; joints [9.124, 53.761, -7.776, -142.234, 52.627, 154.815]
  Call Extruder(707.85487)
  MoveL 10534 to (522.07, 527.3, 192) mm, rotated rx 180 ry 0 rz 160 deg; joints [9.19, 53.67, -7.608, -142.196, 52.715, 154.828]
  Set speed (18.0 mm/s)
  Call Extruder(711.20181)
  MoveL 10535 to (521.23, 527.96, 192) mm, rotated rx 180 ry 0 rz 160 deg; joints [9.284, 53.533, -7.357, -142.142, 52.846, 154.852]
  Call Extruder(714.60272)
  MoveL 10536 to (520.35, 528.6, 192) mm, rotated rx 180 ry 0 rz 160 deg; joints [9.377, 53.389, -7.093, -142.092, 52.98, 154.881]
  Set speed (18.0 mm/s)
  Call Extruder(716.83270)
  MoveL 10537 to (519.77, 529, 192) mm, rotated rx -180 ry 0 rz 160 deg; joints [9.437, 53.293, -6.917, -142.061, 53.069, 154.902]
  Call Extruder(719.16481)
  MoveL 10538 to (519.15, 529.41, 192) mm, rotated rx -180 ry 0 rz 160 deg; joints [9.498, 53.191, -6.729, -142.031, 53.162, 154.926]
  Call Extruder(721.43654)
  MoveL 10539 to (518.54, 529.8, 192) mm, rotated rx -180 ry 0 rz 160 deg; joints [9.556, 53.089, -6.543, -142.004, 53.254, 154.951]
  Set speed (18.0 mm/s)
  Call Extruder(725.94438)
  MoveL 10540 to (517.31, 530.54, 192) mm, rotated rx 180 ry 0 rz 160 deg; joints [9.669, 52.884, -6.166, -141.956, 53.437, 155.007]
  Set speed (18.0 mm/s)
  Call Extruder(728.21860)
  MoveL 10541 to (516.67, 530.89, 192) mm, rotated rx 180 ry 0 rz 160 deg; joints [9.724, 52.778, -5.973, -141.934, 53.529, 155.037]
  Set speed (18.0 mm/s)
  Call Extruder(732.66618)
  MoveL 10542 to (515.41, 531.54, 192) mm, rotated rx -180 ry 0 rz 160 deg; joints [9.827, 52.567, -5.586, -141.897, 53.711, 155.103]
  Set speed (18.0 mm/s)
  Call Extruder(734.88704)
  MoveL 10543 to (514.77, 531.84, 192) mm, rotated rx -180 ry 0 rz 160 deg; joints [9.877, 52.46, -5.389, -141.882, 53.803, 155.139]
  Set speed (18.0 mm/s)
  Call Extruder(739.35050)
  MoveL 10544 to (513.47, 532.41, 192) mm, rotated rx 180 ry 0 rz 160 deg; joints [9.973, 52.241, -4.987, -141.856, 53.986, 155.214]
  Set speed (18.0 mm/s)
  Call Extruder(743.77575)
  MoveL 10545 to (512.15, 532.93, 192) mm, rotated rx 180 ry 0 rz 160 deg; joints [10.063, 52.019, -4.58, -141.838, 54.169, 155.296]
  Set speed (18.0 mm/s)
  Call Extruder(748.32838)
  MoveL 10546 to (510.78, 533.4, 192) mm, rotated rx -180 ry 0 rz 160 deg; joints [10.15, 51.787, -4.155, -141.827, 54.357, 155.387]
  Set speed (18.0 mm/s)
  Call Extruder(752.83209)
  MoveL 10547 to (509.41, 533.81, 192) mm, rotated rx 180 ry 0 rz 160 deg; joints [10.229, 51.553, -3.727, -141.824, 54.543, 155.482]
  Set speed (18.0 mm/s)
  Call Extruder(754.41732)
  MoveL 10548 to (508.92, 533.95, 192) mm, rotated rx -180 ry 0 rz 160 deg; joints [10.256, 51.47, -3.576, -141.824, 54.608, 155.517]
  Call Extruder(757.40352)
  MoveL 10549 to (508, 534.18, 192) mm, rotated rx 180 ry 0 rz 160 deg; joints [10.304, 51.313, -3.288, -141.828, 54.731, 155.585]
  Set speed (18.0 mm/s)
  Call Extruder(761.95060)
  MoveL 10550 to (506.58, 534.48, 192) mm, rotated rx 180 ry 0 rz 160 deg; joints [10.372, 51.07, -2.844, -141.839, 54.917, 155.693]
  Call Extruder(766.52461)
  MoveL 10551 to (505.14, 534.72, 192) mm, rotated rx -180 ry 0 rz 160 deg; joints [10.434, 50.824, -2.393, -141.859, 55.103, 155.808]
  Set speed (18.0 mm/s)
  Call Extruder(770.86963)
  MoveL 10552 to (503.77, 534.9, 192) mm, rotated rx -180 ry 0 rz 160 deg; joints [10.486, 50.587, -1.961, -141.885, 55.278, 155.922]
  Call Extruder(775.49191)
  MoveL 10553 to (502.3, 535.02, 192) mm, rotated rx -180 ry 0 rz 160 deg; joints [10.535, 50.334, -1.499, -141.92, 55.463, 156.048]
  Set speed (18.0 mm/s)
  Call Extruder(780.04939)
  MoveL 10554 to (500.85, 535.09, 192) mm, rotated rx 180 ry 0 rz 160 deg; joints [10.576, 50.083, -1.04, -141.962, 55.643, 156.177]
  Set speed (18.0 mm/s)
  Call Extruder(784.47935)
  MoveL 10555 to (499.43, 535.1, 192) mm, rotated rx 180 ry 0 rz 160 deg; joints [10.61, 49.838, -0.593, -142.01, 55.816, 156.307]
  Set speed (10.0 mm/s)
  MoveL 10556 to (499.43, 535.1, 196) mm, rotated rx -180 ry 0 rz 160 deg; joints [10.61, 49.325, -0.573, -141.801, 55.427, 155.938]
  Set speed (120.0 mm/s)
  MoveL 10557 to (499.43, 535.38, 196) mm, rotated rx 180 ry 0 rz 160 deg; joints [10.644, 49.334, -0.59, -141.76, 55.436, 155.911]
  Set speed (17.9 mm/s)
  Call Extruder(789.10975)
  MoveL 10558 to (497.97, 535.32, 196) mm, rotated rx 180 ry 0 rz 160 deg; joints [10.671, 49.078, -0.125, -141.818, 55.611, 156.051]
  Call Extruder(793.70921)
  MoveL 10559 to (496.52, 535.21, 196) mm, rotated rx -180 ry 0 rz 160 deg; joints [10.692, 48.823, 0.337, -141.883, 55.782, 156.193]
  Set speed (17.9 mm/s)
  Call Extruder(798.20832)
  MoveL 10560 to (495.1, 535.04, 196) mm, rotated rx -180 ry 0 rz 160 deg; joints [10.704, 48.574, 0.789, -141.954, 55.946, 156.336]
  Call Extruder(802.70027)
  MoveL 10561 to (493.7, 534.81, 196) mm, rotated rx -180 ry 0 rz 160 deg; joints [10.709, 48.325, 1.238, -142.033, 56.106, 156.482]
  Call Extruder(807.20297)
  MoveL 10562 to (492.3, 534.53, 196) mm, rotated rx -180 ry 0 rz 160 deg; joints [10.706, 48.077, 1.686, -142.117, 56.263, 156.632]
  Set speed (17.9 mm/s)
  Call Extruder(811.99778)
  MoveL 10563 to (490.83, 534.17, 196) mm, rotated rx 180 ry 0 rz 160 deg; joints [10.696, 47.815, 2.161, -142.215, 56.427, 156.794]
  Set speed (17.9 mm/s)
  Call Extruder(816.34124)
  MoveL 10564 to (489.51, 533.79, 196) mm, rotated rx -180 ry 0 rz 160 deg; joints [10.679, 47.579, 2.587, -142.311, 56.571, 156.944]
  Set speed (17.9 mm/s)
  Call Extruder(821.21503)
  MoveL 10565 to (488.04, 533.3, 196) mm, rotated rx -180 ry 0 rz 160 deg; joints [10.652, 47.317, 3.061, -142.426, 56.728, 157.115]
  Set speed (17.9 mm/s)
  Call Extruder(825.68047)
  MoveL 10566 to (486.72, 532.8, 196) mm, rotated rx -180 ry 0 rz 160 deg; joints [10.62, 47.079, 3.49, -142.538, 56.867, 157.274]
  Set speed (17.8 mm/s)
  Call Extruder(828.83524)
  MoveL 10567 to (485.8, 532.41, 196) mm, rotated rx 180 ry 0 rz 160 deg; joints [10.593, 46.913, 3.79, -142.62, 56.962, 157.387]
  Set speed (17.9 mm/s)
  Call Extruder(832.39523)
  MoveL 10568 to (484.78, 531.94, 196) mm, rotated rx 180 ry 0 rz 160 deg; joints [10.557, 46.727, 4.125, -142.718, 57.067, 157.516]
  Set speed (17.8 mm/s)
  Call Extruder(834.65092)
  MoveL 10569 to (484.14, 531.63, 196) mm, rotated rx -180 ry 0 rz 160 deg; joints [10.533, 46.61, 4.335, -142.782, 57.133, 157.598]
  Call Extruder(837.15146)
  MoveL 10570 to (483.43, 531.26, 196) mm, rotated rx 180 ry 0 rz 160 deg; joints [10.503, 46.482, 4.566, -142.855, 57.203, 157.69]
  Set speed (17.9 mm/s)
  Call Extruder(841.66428)
  MoveL 10571 to (482.18, 530.57, 196) mm, rotated rx -180 ry 0 rz 160 deg; joints [10.443, 46.253, 4.978, -142.991, 57.327, 157.857]
  Set speed (17.9 mm/s)
  Call Extruder(843.90895)
  MoveL 10572 to (481.58, 530.21, 196) mm, rotated rx -180 ry 0 rz 160 deg; joints [10.411, 46.141, 5.179, -143.062, 57.386, 157.94]
  Set speed (17.9 mm/s)
  Call Extruder(846.19180)
  MoveL 10573 to (480.96, 529.82, 196) mm, rotated rx -180 ry 0 rz 160 deg; joints [10.376, 46.028, 5.383, -143.135, 57.445, 158.025]
  Call Extruder(848.46238)
  MoveL 10574 to (480.36, 529.43, 196) mm, rotated rx -180 ry 0 rz 160 deg; joints [10.34, 45.917, 5.583, -143.209, 57.503, 158.11]
  Set speed (17.9 mm/s)
  Call Extruder(850.83404)
  MoveL 10575 to (479.74, 529.01, 196) mm, rotated rx -180 ry 0 rz 160 deg; joints [10.3, 45.802, 5.79, -143.287, 57.562, 158.199]
  Set speed (17.9 mm/s)
  Call Extruder(853.00295)
  MoveL 10576 to (479.18, 528.61, 196) mm, rotated rx 180 ry 0 rz 160 deg; joints [10.261, 45.698, 5.976, -143.361, 57.614, 158.28]
  Set speed (17.9 mm/s)
  Call Extruder(857.68111)
  MoveL 10577 to (478, 527.71, 196) mm, rotated rx 180 ry 0 rz 160 deg; joints [10.173, 45.478, 6.372, -143.525, 57.722, 158.456]
  Set speed (17.9 mm/s)
  Call Extruder(862.11843)
  MoveL 10578 to (476.92, 526.82, 196) mm, rotated rx -180 ry 0 rz 160 deg; joints [10.081, 45.275, 6.737, -143.686, 57.819, 158.623]
  Set speed (17.9 mm/s)
  Call Extruder(864.42014)
  MoveL 10579 to (476.37, 526.34, 196) mm, rotated rx -180 ry 0 rz 160 deg; joints [10.031, 45.171, 6.923, -143.772, 57.867, 158.71]
  Call Extruder(868.03584)
  MoveL 10580 to (475.53, 525.56, 196) mm, rotated rx 180 ry 0 rz 160 deg; joints [9.949, 45.012, 7.209, -143.909, 57.94, 158.846]
  Set speed (17.9 mm/s)
  Call Extruder(871.34171)
  MoveL 10581 to (474.79, 524.82, 196) mm, rotated rx 180 ry 0 rz 160 deg; joints [9.869, 44.87, 7.463, -144.038, 58.002, 158.971]
  Set speed (17.9 mm/s)
  Call Extruder(873.55914)
  MoveL 10582 to (474.3, 524.32, 196) mm, rotated rx 180 ry 0 rz 160 deg; joints [9.814, 44.777, 7.631, -144.126, 58.042, 159.054]
  Set speed (17.9 mm/s)
  Call Extruder(875.87376)
  MoveL 10583 to (473.8, 523.78, 196) mm, rotated rx -180 ry 0 rz 160 deg; joints [9.755, 44.681, 7.803, -144.219, 58.083, 159.141]
  Call Extruder(878.15681)
  MoveL 10584 to (473.32, 523.24, 196) mm, rotated rx -180 ry 0 rz 160 deg; joints [9.695, 44.588, 7.97, -144.312, 58.121, 159.227]
  Call Extruder(880.45657)
  MoveL 10585 to (472.85, 522.68, 196) mm, rotated rx -180 ry 0 rz 160 deg; joints [9.632, 44.496, 8.134, -144.407, 58.158, 159.313]
  Set speed (17.9 mm/s)
  Call Extruder(882.75427)
  MoveL 10586 to (472.39, 522.12, 196) mm, rotated rx -180 ry 0 rz 160 deg; joints [9.568, 44.406, 8.296, -144.504, 58.194, 159.399]
  Set speed (17.9 mm/s)
  Call Extruder(885.01595)
  MoveL 10587 to (471.94, 521.56, 196) mm, rotated rx -180 ry 0 rz 160 deg; joints [9.503, 44.319, 8.451, -144.599, 58.227, 159.484]
  Call Extruder(887.33448)
  MoveL 10588 to (471.5, 520.97, 196) mm, rotated rx -180 ry 0 rz 160 deg; joints [9.435, 44.232, 8.607, -144.699, 58.259, 159.57]
  Call Extruder(891.85157)
  MoveL 10589 to (470.68, 519.8, 196) mm, rotated rx -180 ry 0 rz 160 deg; joints [9.298, 44.068, 8.9, -144.896, 58.317, 159.737]
  Set speed (17.9 mm/s)
  Call Extruder(894.17761)
  MoveL 10590 to (470.27, 519.19, 196) mm, rotated rx -180 ry 0 rz 160 deg; joints [9.225, 43.987, 9.046, -145, 58.345, 159.823]
  Call Extruder(896.46414)
  MoveL 10591 to (469.89, 518.57, 196) mm, rotated rx -180 ry 0 rz 160 deg; joints [9.152, 43.909, 9.186, -145.102, 58.37, 159.907]
  Set speed (17.9 mm/s)
  Call Extruder(898.76954)
  MoveL 10592 to (469.51, 517.95, 196) mm, rotated rx 180 ry 0 rz 160 deg; joints [9.077, 43.832, 9.323, -145.207, 58.394, 159.991]
  Set speed (17.9 mm/s)
  Call Extruder(900.95659)
  MoveL 10593 to (469.16, 517.35, 196) mm, rotated rx 180 ry 0 rz 160 deg; joints [9.004, 43.761, 9.45, -145.307, 58.415, 160.07]
  Set speed (17.9 mm/s)
  Call Extruder(903.40486)
  MoveL 10594 to (468.79, 516.67, 196) mm, rotated rx -180 ry 0 rz 160 deg; joints [8.921, 43.684, 9.588, -145.419, 58.437, 160.159]
  Set speed (17.9 mm/s)
  Call Extruder(907.99626)
  MoveL 10595 to (468.13, 515.37, 196) mm, rotated rx -180 ry 0 rz 160 deg; joints [8.761, 43.546, 9.834, -145.633, 58.472, 160.323]
  Set speed (17.9 mm/s)
  Call Extruder(912.43422)
  MoveL 10596 to (467.55, 514.1, 196) mm, rotated rx 180 ry 0 rz 160 deg; joints [8.602, 43.422, 10.057, -145.844, 58.5, 160.48]
  Call Extruder(916.95095)
  MoveL 10597 to (467, 512.77, 196) mm, rotated rx -180 ry 0 rz 160 deg; joints [8.435, 43.303, 10.269, -146.06, 58.522, 160.638]
  Set speed (17.9 mm/s)
  Call Extruder(921.69256)
  MoveL 10598 to (466.49, 511.36, 196) mm, rotated rx 180 ry 0 rz 160 deg; joints [8.255, 43.188, 10.474, -146.29, 58.537, 160.801]
  Call Extruder(926.11334)
  MoveL 10599 to (466.07, 510.03, 196) mm, rotated rx -180 ry 0 rz 160 deg; joints [8.083, 43.09, 10.649, -146.507, 58.545, 160.95]
  Set speed (17.9 mm/s)
  Call Extruder(930.68801)
  MoveL 10600 to (465.69, 508.63, 196) mm, rotated rx -180 ry 0 rz 160 deg; joints [7.901, 42.998, 10.812, -146.733, 58.546, 161.102]
  Set speed (17.9 mm/s)
  Call Extruder(935.20120)
  MoveL 10601 to (465.37, 507.24, 196) mm, rotated rx 180 ry 0 rz 160 deg; joints [7.718, 42.917, 10.957, -146.957, 58.54, 161.248]
  Set speed (17.9 mm/s)
  Call Extruder(939.98012)
  MoveL 10602 to (465.09, 505.75, 196) mm, rotated rx -180 ry 0 rz 160 deg; joints [7.521, 42.841, 11.093, -147.195, 58.527, 161.401]
  Set speed (17.9 mm/s)
  Call Extruder(944.55874)
  MoveL 10603 to (464.88, 504.32, 196) mm, rotated rx 180 ry 0 rz 160 deg; joints [7.329, 42.779, 11.204, -147.425, 58.507, 161.543]
  Call Extruder(949.13534)
  MoveL 10604 to (464.74, 502.87, 196) mm, rotated rx -180 ry 0 rz 160 deg; joints [7.136, 42.726, 11.299, -147.654, 58.481, 161.681]
  Set speed (17.9 mm/s)
  Call Extruder(953.66005)
  MoveL 10605 to (464.65, 501.44, 196) mm, rotated rx -180 ry 0 rz 160 deg; joints [6.942, 42.684, 11.374, -147.88, 58.448, 161.815]
  Set speed (17.8 mm/s)
  Call Extruder(958.14954)
  MoveL 10606 to (464.62, 500.03, 196) mm, rotated rx -180 ry 0 rz 160 deg; joints [6.749, 42.653, 11.429, -148.103, 58.409, 161.943]
  Set speed (17.8 mm/s)
  Call Extruder(962.23151)
  MoveL 10607 to (464.64, 498.74, 196) mm, rotated rx 180 ry 0 rz 160 deg; joints [6.573, 42.632, 11.466, -148.306, 58.368, 162.056]
  Set speed (17.9 mm/s)
  Call Extruder(966.42607)
  MoveL 10608 to (464.71, 497.41, 196) mm, rotated rx 180 ry 0 rz 160 deg; joints [6.39, 42.619, 11.489, -148.513, 58.321, 162.169]
  Set speed (17.9 mm/s)
  Call Extruder(970.65798)
  MoveL 10609 to (464.84, 496.07, 196) mm, rotated rx 180 ry 0 rz 160 deg; joints [6.206, 42.616, 11.495, -148.72, 58.267, 162.279]
  Set speed (17.9 mm/s)
  Call Extruder(974.65572)
  MoveL 10610 to (465, 494.82, 196) mm, rotated rx -180 ry 0 rz 160 deg; joints [6.032, 42.62, 11.487, -148.914, 58.211, 162.38]
  Call Extruder(978.86016)
  MoveL 10611 to (465.22, 493.51, 196) mm, rotated rx -180 ry 0 rz 160 deg; joints [5.849, 42.633, 11.464, -149.116, 58.147, 162.482]
  Set speed (17.9 mm/s)
  Call Extruder(983.10601)
  MoveL 10612 to (465.49, 492.19, 196) mm, rotated rx -180 ry 0 rz 160 deg; joints [5.666, 42.655, 11.424, -149.317, 58.077, 162.58]
  Set speed (17.9 mm/s)
  Call Extruder(987.04715)
  MoveL 10613 to (465.79, 490.98, 196) mm, rotated rx 180 ry 0 rz 160 deg; joints [5.496, 42.684, 11.373, -149.5, 58.007, 162.668]
  Set speed (17.9 mm/s)
  Call Extruder(991.03445)
  MoveL 10614 to (466.13, 489.77, 196) mm, rotated rx 180 ry 0 rz 160 deg; joints [5.325, 42.72, 11.309, -149.683, 57.932, 162.753]
  Set speed (17.9 mm/s)
  Call Extruder(995.15765)
  MoveL 10615 to (466.53, 488.52, 196) mm, rotated rx -180 ry 0 rz 160 deg; joints [5.15, 42.766, 11.227, -149.869, 57.849, 162.836]
  Set speed (17.9 mm/s)
  Call Extruder(999.38294)
  MoveL 10616 to (466.99, 487.26, 196) mm, rotated rx -180 ry 0 rz 160 deg; joints [4.973, 42.821, 11.128, -150.056, 57.759, 162.917]
  Set speed (17.9 mm/s)
  Call Extruder(1002.57299)
  MoveL 10617 to (467.37, 486.33, 196) mm, rotated rx 180 ry 0 rz 160 deg; joints [4.841, 42.868, 11.044, -150.194, 57.689, 162.976]
  Set speed (17.9 mm/s)
  Call Extruder(1007.53749)
  MoveL 10618 to (468, 484.89, 196) mm, rotated rx 180 ry 0 rz 160 deg; joints [4.638, 42.952, 10.895, -150.403, 57.572, 163.06]
  Set speed (17.9 mm/s)
  Call Extruder(1011.71374)
  MoveL 10619 to (468.59, 483.71, 196) mm, rotated rx 180 ry 0 rz 160 deg; joints [4.47, 43.031, 10.755, -150.574, 57.47, 163.126]
  Set speed (17.9 mm/s)
  Call Extruder(1015.78815)
  MoveL 10620 to (469.21, 482.58, 196) mm, rotated rx 180 ry 0 rz 160 deg; joints [4.309, 43.115, 10.604, -150.736, 57.365, 163.186]
  Set speed (17.9 mm/s)
  Call Extruder(1019.95560)
  MoveL 10621 to (469.88, 481.44, 196) mm, rotated rx 180 ry 0 rz 160 deg; joints [4.148, 43.21, 10.434, -150.896, 57.254, 163.242]
  Set speed (17.9 mm/s)
  Call Extruder(1023.96906)
  MoveL 10622 to (470.57, 480.37, 196) mm, rotated rx -180 ry 0 rz 160 deg; joints [3.996, 43.308, 10.259, -151.045, 57.143, 163.291]
  Set speed (17.9 mm/s)
  Call Extruder(1028.14100)
  MoveL 10623 to (471.32, 479.29, 196) mm, rotated rx 180 ry 0 rz 160 deg; joints [3.842, 43.418, 10.064, -151.195, 57.023, 163.338]
  Set speed (17.9 mm/s)
  Call Extruder(1032.12597)
  MoveL 10624 to (472.08, 478.28, 196) mm, rotated rx 180 ry 0 rz 160 deg; joints [3.698, 43.529, 9.864, -151.331, 56.905, 163.377]
  Set speed (17.9 mm/s)
  Call Extruder(1036.31693)
  MoveL 10625 to (472.91, 477.24, 196) mm, rotated rx -180 ry 0 rz 160 deg; joints [3.551, 43.654, 9.642, -151.468, 56.777, 163.412]
  Call Extruder(1040.47242)
  MoveL 10626 to (473.77, 476.25, 196) mm, rotated rx 180 ry 0 rz 160 deg; joints [3.41, 43.784, 9.409, -151.598, 56.646, 163.443]
  Set speed (17.9 mm/s)
  Call Extruder(1044.66813)
  MoveL 10627 to (474.69, 475.28, 196) mm, rotated rx 180 ry 0 rz 160 deg; joints [3.272, 43.923, 9.161, -151.722, 56.511, 163.468]
  Set speed (17.9 mm/s)
  Call Extruder(1048.74451)
  MoveL 10628 to (475.6, 474.38, 196) mm, rotated rx 180 ry 0 rz 160 deg; joints [3.143, 44.064, 8.908, -151.836, 56.376, 163.486]
  Set speed (17.9 mm/s)
  Call Extruder(1052.66220)
  MoveL 10629 to (476.52, 473.54, 196) mm, rotated rx -180 ry 0 rz 160 deg; joints [3.024, 44.206, 8.654, -151.938, 56.243, 163.499]
  Set speed (17.9 mm/s)
  Call Extruder(1057.00440)
  MoveL 10630 to (477.56, 472.64, 196) mm, rotated rx 180 ry 0 rz 160 deg; joints [2.897, 44.369, 8.362, -152.044, 56.093, 163.508]
  Call Extruder(1061.04096)
  MoveL 10631 to (478.57, 471.85, 196) mm, rotated rx -180 ry 0 rz 160 deg; joints [2.784, 44.527, 8.079, -152.135, 55.951, 163.51]
  Set speed (17.9 mm/s)
  Call Extruder(1065.24804)
  MoveL 10632 to (479.64, 471.06, 196) mm, rotated rx -180 ry 0 rz 160 deg; joints [2.672, 44.697, 7.774, -152.222, 55.8, 163.507]
  Set speed (17.9 mm/s)
  Call Extruder(1069.25464)
  MoveL 10633 to (480.69, 470.35, 196) mm, rotated rx -180 ry 0 rz 160 deg; joints [2.571, 44.865, 7.473, -152.297, 55.653, 163.498]
  Set speed (17.9 mm/s)
  Call Extruder(1073.46566)
  MoveL 10634 to (481.82, 469.65, 196) mm, rotated rx 180 ry 0 rz 160 deg; joints [2.471, 45.047, 7.147, -152.367, 55.497, 163.482]
  Set speed (17.9 mm/s)
  Call Extruder(1077.58196)
  MoveL 10635 to (482.95, 469, 196) mm, rotated rx -180 ry 0 rz 160 deg; joints [2.379, 45.229, 6.82, -152.429, 55.342, 163.462]
  Set speed (17.9 mm/s)
  Call Extruder(1082.53767)
  MoveL 10636 to (484.34, 468.27, 196) mm, rotated rx -180 ry 0 rz 160 deg; joints [2.275, 45.455, 6.414, -152.492, 55.153, 163.43]
  Set speed (17.9 mm/s)
  Call Extruder(1085.64319)
  MoveL 10637 to (485.23, 467.85, 196) mm, rotated rx -180 ry 0 rz 160 deg; joints [2.215, 45.6, 6.153, -152.524, 55.033, 163.405]
  Set speed (17.9 mm/s)
  Call Extruder(1089.99442)
  MoveL 10638 to (486.49, 467.3, 196) mm, rotated rx 180 ry 0 rz 160 deg; joints [2.136, 45.807, 5.781, -152.563, 54.864, 163.364]
  Set speed (17.9 mm/s)
  Call Extruder(1093.90166)
  MoveL 10639 to (487.64, 466.85, 196) mm, rotated rx -180 ry 0 rz 160 deg; joints [2.072, 45.997, 5.439, -152.59, 54.711, 163.323]
  Call Extruder(1098.15896)
  MoveL 10640 to (488.91, 466.4, 196) mm, rotated rx -180 ry 0 rz 160 deg; joints [2.007, 46.208, 5.059, -152.611, 54.543, 163.271]
  Set speed (17.9 mm/s)
  Call Extruder(1102.14351)
  MoveL 10641 to (490.12, 466.03, 196) mm, rotated rx 180 ry 0 rz 160 deg; joints [1.953, 46.409, 4.697, -152.621, 54.384, 163.217]
  Set speed (17.9 mm/s)
  Call Extruder(1106.16276)
  MoveL 10642 to (491.35, 465.69, 196) mm, rotated rx -180 ry 0 rz 160 deg; joints [1.904, 46.615, 4.327, -152.624, 54.224, 163.157]
  Set speed (17.9 mm/s)
  Call Extruder(1110.49040)
  MoveL 10643 to (492.68, 465.38, 196) mm, rotated rx 180 ry 0 rz 160 deg; joints [1.859, 46.84, 3.922, -152.618, 54.05, 163.087]
  Call Extruder(1114.47989)
  MoveL 10644 to (493.92, 465.15, 196) mm, rotated rx 180 ry 0 rz 160 deg; joints [1.823, 47.049, 3.543, -152.604, 53.89, 163.016]
  Set speed (17.9 mm/s)
  Call Extruder(1118.30457)
  MoveL 10645 to (495.12, 464.96, 196) mm, rotated rx -180 ry 0 rz 160 deg; joints [1.793, 47.253, 3.176, -152.584, 53.736, 162.943]
  Set speed (17.9 mm/s)
  Call Extruder(1122.79971)
  MoveL 10646 to (496.53, 464.79, 196) mm, rotated rx 180 ry 0 rz 160 deg; joints [1.766, 47.494, 2.741, -152.55, 53.556, 162.851]
  Call Extruder(1126.79062)
  MoveL 10647 to (497.79, 464.69, 196) mm, rotated rx -180 ry 0 rz 160 deg; joints [1.748, 47.71, 2.35, -152.512, 53.396, 162.764]
  Set speed (17.9 mm/s)
  Call Extruder(1131.06785)
  MoveL 10648 to (499.14, 464.63, 196) mm, rotated rx -180 ry 0 rz 160 deg; joints [1.736, 47.943, 1.928, -152.462, 53.225, 162.664]
  Set speed (17.9 mm/s)
  Call Extruder(1135.10578)
  MoveL 10649 to (500.42, 464.62, 196) mm, rotated rx 180 ry 0 rz 160 deg; joints [1.73, 48.165, 1.528, -152.407, 53.064, 162.565]
  Set speed (17.9 mm/s)
  Call Extruder(1139.28910)
  MoveL 10650 to (501.75, 464.66, 196) mm, rotated rx 180 ry 0 rz 160 deg; joints [1.73, 48.396, 1.11, -152.342, 52.899, 162.456]
  Set speed (17.9 mm/s)
  Call Extruder(1143.33680)
  MoveL 10651 to (503.03, 464.75, 196) mm, rotated rx 180 ry 0 rz 160 deg; joints [1.736, 48.62, 0.704, -152.271, 52.74, 162.346]
  Set speed (17.9 mm/s)
  Call Extruder(1147.52350)
  MoveL 10652 to (504.35, 464.89, 196) mm, rotated rx -180 ry 0 rz 160 deg; joints [1.748, 48.852, 0.284, -152.189, 52.577, 162.227]
  Set speed (17.9 mm/s)
  Call Extruder(1151.47468)
  MoveL 10653 to (505.59, 465.06, 196) mm, rotated rx -180 ry 0 rz 160 deg; joints [1.765, 49.071, -0.113, -152.104, 52.425, 162.109]
  Set speed (17.9 mm/s)
  Call Extruder(1155.54511)
  MoveL 10654 to (506.86, 465.29, 196) mm, rotated rx 180 ry 0 rz 160 deg; joints [1.789, 49.297, -0.522, -152.01, 52.27, 161.983]
  Set speed (17.9 mm/s)
  Call Extruder(1159.09084)
  MoveL 10655 to (507.95, 465.52, 196) mm, rotated rx -180 ry 0 rz 160 deg; joints [1.814, 49.493, -0.878, -151.921, 52.137, 161.87]
  Set speed (17.9 mm/s)
  Call Extruder(1163.83123)
  MoveL 10656 to (509.41, 465.89, 196) mm, rotated rx 180 ry 0 rz 160 deg; joints [1.854, 49.754, -1.352, -151.795, 51.962, 161.713]
  Set speed (17.9 mm/s)
  Call Extruder(1168.02391)
  MoveL 10657 to (510.68, 466.27, 196) mm, rotated rx 180 ry 0 rz 160 deg; joints [1.896, 49.984, -1.77, -151.675, 51.81, 161.569]
  Set speed (17.9 mm/s)
  Call Extruder(1172.19087)
  MoveL 10658 to (511.93, 466.69, 196) mm, rotated rx 180 ry 0 rz 160 deg; joints [1.943, 50.212, -2.182, -151.548, 51.662, 161.421]
  Set speed (17.9 mm/s)
  Call Extruder(1176.22191)
  MoveL 10659 to (513.13, 467.14, 196) mm, rotated rx 180 ry 0 rz 160 deg; joints [1.994, 50.43, -2.579, -151.419, 51.521, 161.274]
  Call Extruder(1180.41423)
  MoveL 10660 to (514.35, 467.66, 196) mm, rotated rx 180 ry 0 rz 160 deg; joints [2.053, 50.655, -2.988, -151.278, 51.379, 161.118]
  Set speed (17.9 mm/s)
  Call Extruder(1184.44330)
  MoveL 10661 to (515.51, 468.2, 196) mm, rotated rx 180 ry 0 rz 160 deg; joints [2.114, 50.869, -3.377, -151.136, 51.245, 160.963]
  Call Extruder(1188.65173)
  MoveL 10662 to (516.69, 468.81, 196) mm, rotated rx 180 ry 0 rz 160 deg; joints [2.183, 51.09, -3.779, -150.982, 51.109, 160.798]
  Set speed (17.9 mm/s)
  Call Extruder(1192.76161)
  MoveL 10663 to (517.83, 469.44, 196) mm, rotated rx 180 ry 0 rz 160 deg; joints [2.255, 51.303, -4.167, -150.825, 50.98, 160.633]
  Set speed (17.9 mm/s)
  Call Extruder(1196.78259)
  MoveL 10664 to (518.92, 470.1, 196) mm, rotated rx -180 ry 0 rz 160 deg; joints [2.331, 51.508, -4.541, -150.667, 50.858, 160.469]
  Set speed (17.9 mm/s)
  Call Extruder(1200.97849)
  MoveL 10665 to (520.03, 470.83, 196) mm, rotated rx 180 ry 0 rz 160 deg; joints [2.415, 51.719, -4.925, -150.495, 50.736, 160.295]
  Call Extruder(1204.86541)
  MoveL 10666 to (521.03, 471.55, 196) mm, rotated rx -180 ry 0 rz 160 deg; joints [2.496, 51.911, -5.275, -150.332, 50.626, 160.132]
  Call Extruder(1209.12101)
  MoveL 10667 to (522.1, 472.37, 196) mm, rotated rx 180 ry 0 rz 160 deg; joints [2.59, 52.117, -5.65, -150.148, 50.511, 159.95]
  Call Extruder(1213.23555)
  MoveL 10668 to (523.1, 473.2, 196) mm, rotated rx 180 ry 0 rz 160 deg; joints [2.686, 52.312, -6.005, -149.966, 50.405, 159.772]
  Set speed (17.9 mm/s)
  Call Extruder(1217.44704)
  MoveL 10669 to (524.09, 474.09, 196) mm, rotated rx -180 ry 0 rz 160 deg; joints [2.788, 52.506, -6.36, -149.775, 50.301, 159.588]
  Set speed (17.9 mm/s)
  Call Extruder(1221.40378)
  MoveL 10670 to (525, 474.96, 196) mm, rotated rx 180 ry 0 rz 160 deg; joints [2.887, 52.685, -6.686, -149.593, 50.209, 159.414]
  Set speed (17.9 mm/s)
  Call Extruder(1226.09580)
  MoveL 10671 to (526.03, 476.03, 196) mm, rotated rx -180 ry 0 rz 160 deg; joints [3.009, 52.89, -7.061, -149.372, 50.106, 159.207]
  Set speed (17.9 mm/s)
  Call Extruder(1230.45391)
  MoveL 10672 to (526.94, 477.06, 196) mm, rotated rx 180 ry 0 rz 160 deg; joints [3.128, 53.075, -7.398, -149.162, 50.017, 159.012]
  Call Extruder(1232.86379)
  MoveL 10673 to (527.43, 477.65, 196) mm, rotated rx 180 ry 0 rz 160 deg; joints [3.195, 53.174, -7.579, -149.045, 49.971, 158.905]
  Set speed (17.9 mm/s)
  Call Extruder(1235.20042)
  MoveL 10674 to (527.89, 478.23, 196) mm, rotated rx 180 ry 0 rz 160 deg; joints [3.261, 53.268, -7.752, -148.931, 49.928, 158.8]
  Set speed (17.9 mm/s)
  Call Extruder(1239.75361)
  MoveL 10675 to (528.75, 479.39, 196) mm, rotated rx -180 ry 0 rz 160 deg; joints [3.393, 53.446, -8.078, -148.705, 49.85, 158.597]
  Set speed (17.9 mm/s)
  Call Extruder(1242.08233)
  MoveL 10676 to (529.18, 479.99, 196) mm, rotated rx 180 ry 0 rz 160 deg; joints [3.462, 53.535, -8.24, -148.589, 49.812, 158.493]
  Set speed (17.9 mm/s)
  Call Extruder(1244.24945)
  MoveL 10677 to (529.56, 480.56, 196) mm, rotated rx 180 ry 0 rz 160 deg; joints [3.527, 53.615, -8.386, -148.48, 49.78, 158.396]
  Call Extruder(1246.50441)
  MoveL 10678 to (529.95, 481.16, 196) mm, rotated rx -180 ry 0 rz 160 deg; joints [3.596, 53.697, -8.536, -148.367, 49.747, 158.296]
  Set speed (17.9 mm/s)
  Call Extruder(1248.83133)
  MoveL 10679 to (530.33, 481.79, 196) mm, rotated rx 180 ry 0 rz 160 deg; joints [3.668, 53.779, -8.686, -148.249, 49.716, 158.192]
  Set speed (17.9 mm/s)
  Call Extruder(1251.10018)
  MoveL 10680 to (530.7, 482.41, 196) mm, rotated rx -180 ry 0 rz 160 deg; joints [3.739, 53.857, -8.829, -148.134, 49.687, 158.092]
  Set speed (17.8 mm/s)
  Call Extruder(1254.72222)
  MoveL 10681 to (531.25, 483.41, 196) mm, rotated rx -180 ry 0 rz 160 deg; joints [3.853, 53.978, -9.049, -147.95, 49.645, 157.932]
  Set speed (17.8 mm/s)
  Call Extruder(1258.07194)
  MoveL 10682 to (531.73, 484.35, 196) mm, rotated rx 180 ry 0 rz 160 deg; joints [3.961, 54.083, -9.242, -147.779, 49.612, 157.786]
  Set speed (17.8 mm/s)
  Call Extruder(1261.37557)
  MoveL 10683 to (532.18, 485.29, 196) mm, rotated rx 180 ry 0 rz 160 deg; joints [4.069, 54.184, -9.427, -147.61, 49.582, 157.642]
  Set speed (17.9 mm/s)
  Call Extruder(1267.02448)
  MoveL 10684 to (532.88, 486.94, 196) mm, rotated rx 180 ry 0 rz 160 deg; joints [4.257, 54.344, -9.72, -147.32, 49.542, 157.4]
  Set speed (17.9 mm/s)
  Call Extruder(1271.77323)
  MoveL 10685 to (533.41, 488.35, 196) mm, rotated rx -180 ry 0 rz 160 deg; joints [4.419, 54.467, -9.946, -147.077, 49.518, 157.2]
  Set speed (17.9 mm/s)
  Call Extruder(1276.28374)
  MoveL 10686 to (533.85, 489.7, 196) mm, rotated rx -180 ry 0 rz 160 deg; joints [4.575, 54.575, -10.143, -146.846, 49.504, 157.013]
  Set speed (17.9 mm/s)
  Call Extruder(1280.84015)
  MoveL 10687 to (534.24, 491.09, 196) mm, rotated rx -180 ry 0 rz 160 deg; joints [4.735, 54.675, -10.325, -146.614, 49.497, 156.828]
  Set speed (17.9 mm/s)
  Call Extruder(1285.37610)
  MoveL 10688 to (534.58, 492.49, 196) mm, rotated rx -180 ry 0 rz 160 deg; joints [4.896, 54.764, -10.488, -146.384, 49.499, 156.647]
  Call Extruder(1290.03402)
  MoveL 10689 to (534.86, 493.94, 196) mm, rotated rx -180 ry 0 rz 160 deg; joints [5.063, 54.844, -10.636, -146.151, 49.51, 156.467]
  Set speed (17.9 mm/s)
  Call Extruder(1294.51464)
  MoveL 10690 to (535.07, 495.34, 196) mm, rotated rx -180 ry 0 rz 160 deg; joints [5.226, 54.912, -10.759, -145.928, 49.529, 156.299]
  Set speed (17.9 mm/s)
  Call Extruder(1299.25844)
  MoveL 10691 to (535.24, 496.83, 196) mm, rotated rx 180 ry 0 rz 160 deg; joints [5.399, 54.972, -10.87, -145.696, 49.557, 156.127]
  Call Extruder(1303.72485)
  MoveL 10692 to (535.34, 498.25, 196) mm, rotated rx 180 ry 0 rz 160 deg; joints [5.563, 55.019, -10.955, -145.48, 49.592, 155.97]
  Set speed (17.9 mm/s)
  Call Extruder(1308.31286)
  MoveL 10693 to (535.38, 499.7, 196) mm, rotated rx -180 ry 0 rz 160 deg; joints [5.733, 55.055, -11.022, -145.262, 49.636, 155.816]
  Set speed (17.9 mm/s)
  Call Extruder(1312.75506)
  MoveL 10694 to (535.36, 501.11, 196) mm, rotated rx 180 ry 0 rz 160 deg; joints [5.898, 55.081, -11.069, -145.055, 49.686, 155.672]
  Set speed (17.9 mm/s)
  Call Extruder(1317.43125)
  MoveL 10695 to (535.29, 502.58, 196) mm, rotated rx -180 ry 0 rz 160 deg; joints [6.072, 55.096, -11.098, -144.841, 49.747, 155.528]
  Set speed (17.9 mm/s)
  Call Extruder(1321.93641)
  MoveL 10696 to (535.15, 504.01, 196) mm, rotated rx 180 ry 0 rz 160 deg; joints [6.239, 55.1, -11.105, -144.639, 49.814, 155.397]
  Set speed (17.9 mm/s)
  Call Extruder(1326.67487)
  MoveL 10697 to (534.95, 505.49, 196) mm, rotated rx -180 ry 0 rz 160 deg; joints [6.416, 55.093, -11.092, -144.432, 49.893, 155.266]
  Set speed (17.9 mm/s)
  Call Extruder(1331.23177)
  MoveL 10698 to (534.7, 506.92, 196) mm, rotated rx 180 ry 0 rz 160 deg; joints [6.585, 55.075, -11.058, -144.239, 49.976, 155.148]
  Set speed (17.9 mm/s)
  Call Extruder(1336.09176)
  MoveL 10699 to (534.37, 508.42, 196) mm, rotated rx -180 ry 0 rz 160 deg; joints [6.765, 55.044, -11.002, -144.038, 50.073, 155.031]
  Set speed (17.9 mm/s)
  Call Extruder(1340.19562)
  MoveL 10700 to (534.03, 509.67, 196) mm, rotated rx 180 ry 0 rz 160 deg; joints [6.917, 55.008, -10.936, -143.874, 50.161, 154.939]
  Set speed (17.9 mm/s)
  Call Extruder(1344.71945)
  MoveL 10701 to (533.61, 511.04, 196) mm, rotated rx -180 ry 0 rz 160 deg; joints [7.083, 54.958, -10.845, -143.699, 50.265, 154.846]
  Set speed (17.9 mm/s)
  Call Extruder(1349.34627)
  MoveL 10702 to (533.13, 512.43, 196) mm, rotated rx 180 ry 0 rz 160 deg; joints [7.251, 54.896, -10.731, -143.526, 50.378, 154.759]
  Set speed (17.9 mm/s)
  Call Extruder(1354.17888)
  MoveL 10703 to (532.56, 513.85, 196) mm, rotated rx -180 ry 0 rz 160 deg; joints [7.426, 54.821, -10.593, -143.352, 50.503, 154.677]
  Set speed (17.8 mm/s)
  Call Extruder(1359.43213)
  MoveL 10704 to (531.88, 515.36, 196) mm, rotated rx -180 ry 0 rz 160 deg; joints [7.614, 54.726, -10.419, -143.171, 50.647, 154.599]
  Call Extruder(1363.06504)
  MoveL 10705 to (531.36, 516.39, 196) mm, rotated rx -180 ry 0 rz 160 deg; joints [7.742, 54.652, -10.283, -143.052, 50.752, 154.552]
  Set speed (17.9 mm/s)
  Call Extruder(1367.63372)
  MoveL 10706 to (530.66, 517.65, 196) mm, rotated rx 180 ry 0 rz 160 deg; joints [7.902, 54.55, -10.096, -142.907, 50.888, 154.5]
  Call Extruder(1369.92827)
  MoveL 10707 to (530.29, 518.28, 196) mm, rotated rx -180 ry 0 rz 160 deg; joints [7.981, 54.495, -9.996, -142.838, 50.958, 154.478]
  Call Extruder(1374.50384)
  MoveL 10708 to (529.52, 519.51, 196) mm, rotated rx 180 ry 0 rz 160 deg; joints [8.137, 54.378, -9.782, -142.704, 51.103, 154.439]
  Set speed (17.9 mm/s)
  Call Extruder(1379.04889)
  MoveL 10709 to (528.7, 520.69, 196) mm, rotated rx 180 ry 0 rz 160 deg; joints [8.29, 54.252, -9.552, -142.578, 51.252, 154.409]
  Set speed (17.9 mm/s)
  Call Extruder(1381.39485)
  MoveL 10710 to (528.26, 521.29, 196) mm, rotated rx -180 ry 0 rz 160 deg; joints [8.368, 54.184, -9.427, -142.515, 51.331, 154.397]
  Call Extruder(1383.76103)
  MoveL 10711 to (527.8, 521.88, 196) mm, rotated rx -180 ry 0 rz 160 deg; joints [8.446, 54.113, -9.297, -142.454, 51.411, 154.387]
  Set speed (17.9 mm/s)
  Call Extruder(1385.96991)
  MoveL 10712 to (527.37, 522.43, 196) mm, rotated rx 180 ry 0 rz 160 deg; joints [8.518, 54.044, -9.17, -142.399, 51.488, 154.38]
  Set speed (17.9 mm/s)
  Call Extruder(1388.27401)
  MoveL 10713 to (526.9, 522.99, 196) mm, rotated rx -180 ry 0 rz 160 deg; joints [8.592, 53.97, -9.035, -142.344, 51.568, 154.375]
  Set speed (17.9 mm/s)
  Call Extruder(1390.53916)
  MoveL 10714 to (526.42, 523.53, 196) mm, rotated rx -180 ry 0 rz 160 deg; joints [8.664, 53.895, -8.898, -142.291, 51.649, 154.372]
  Set speed (17.9 mm/s)
  Call Extruder(1392.82260)
  MoveL 10715 to (525.94, 524.06, 196) mm, rotated rx 180 ry 0 rz 160 deg; joints [8.735, 53.818, -8.757, -142.24, 51.73, 154.371]
  Set speed (17.9 mm/s)
  Call Extruder(1397.38263)
  MoveL 10716 to (524.93, 525.1, 196) mm, rotated rx -180 ry 0 rz 160 deg; joints [8.876, 53.656, -8.462, -142.143, 51.897, 154.375]
  Set speed (17.9 mm/s)
  Call Extruder(1401.83872)
  MoveL 10717 to (523.91, 526.08, 196) mm, rotated rx -180 ry 0 rz 160 deg; joints [9.01, 53.491, -8.16, -142.055, 52.063, 154.388]
  Set speed (17.9 mm/s)
  Call Extruder(1406.11919)
  MoveL 10718 to (522.9, 526.97, 196) mm, rotated rx 180 ry 0 rz 160 deg; joints [9.135, 53.326, -7.857, -141.978, 52.225, 154.407]
  Call Extruder(1408.79580)
  MoveL 10719 to (522.24, 527.51, 196) mm, rotated rx 180 ry 0 rz 160 deg; joints [9.212, 53.218, -7.661, -141.933, 52.328, 154.423]
  Set speed (17.9 mm/s)
  Call Extruder(1413.36181)
  MoveL 10720 to (521.1, 528.4, 196) mm, rotated rx -180 ry 0 rz 160 deg; joints [9.339, 53.031, -7.318, -141.862, 52.505, 154.455]
  Set speed (17.9 mm/s)
  Call Extruder(1415.60284)
  MoveL 10721 to (520.53, 528.82, 196) mm, rotated rx -180 ry 0 rz 160 deg; joints [9.4, 52.936, -7.145, -141.83, 52.593, 154.474]
  Set speed (17.9 mm/s)
  Call Extruder(1417.92493)
  MoveL 10722 to (519.92, 529.24, 196) mm, rotated rx -180 ry 0 rz 160 deg; joints [9.462, 52.836, -6.962, -141.798, 52.684, 154.496]
  Set speed (17.9 mm/s)
  Call Extruder(1420.26104)
  MoveL 10723 to (519.31, 529.65, 196) mm, rotated rx -180 ry 0 rz 160 deg; joints [9.523, 52.733, -6.775, -141.769, 52.777, 154.52]
  Set speed (17.9 mm/s)
  Call Extruder(1422.47806)
  MoveL 10724 to (518.72, 530.03, 196) mm, rotated rx 180 ry 0 rz 160 deg; joints [9.579, 52.635, -6.595, -141.743, 52.865, 154.544]
  Set speed (17.9 mm/s)
  Call Extruder(1424.84877)
  MoveL 10725 to (518.07, 530.41, 196) mm, rotated rx 180 ry 0 rz 160 deg; joints [9.638, 52.527, -6.399, -141.718, 52.96, 154.572]
  Set speed (17.9 mm/s)
  Call Extruder(1428.84534)
  MoveL 10726 to (516.98, 531.04, 196) mm, rotated rx -180 ry 0 rz 160 deg; joints [9.736, 52.344, -6.065, -141.678, 53.121, 154.624]
  Set speed (17.9 mm/s)
  Call Extruder(1431.48907)
